REGION Network 26: *** 8 - Outputs *** Status
   #O_Status := #Status;
END_REGION

REGION Network 27: *** 8 - Outputs *** Busy
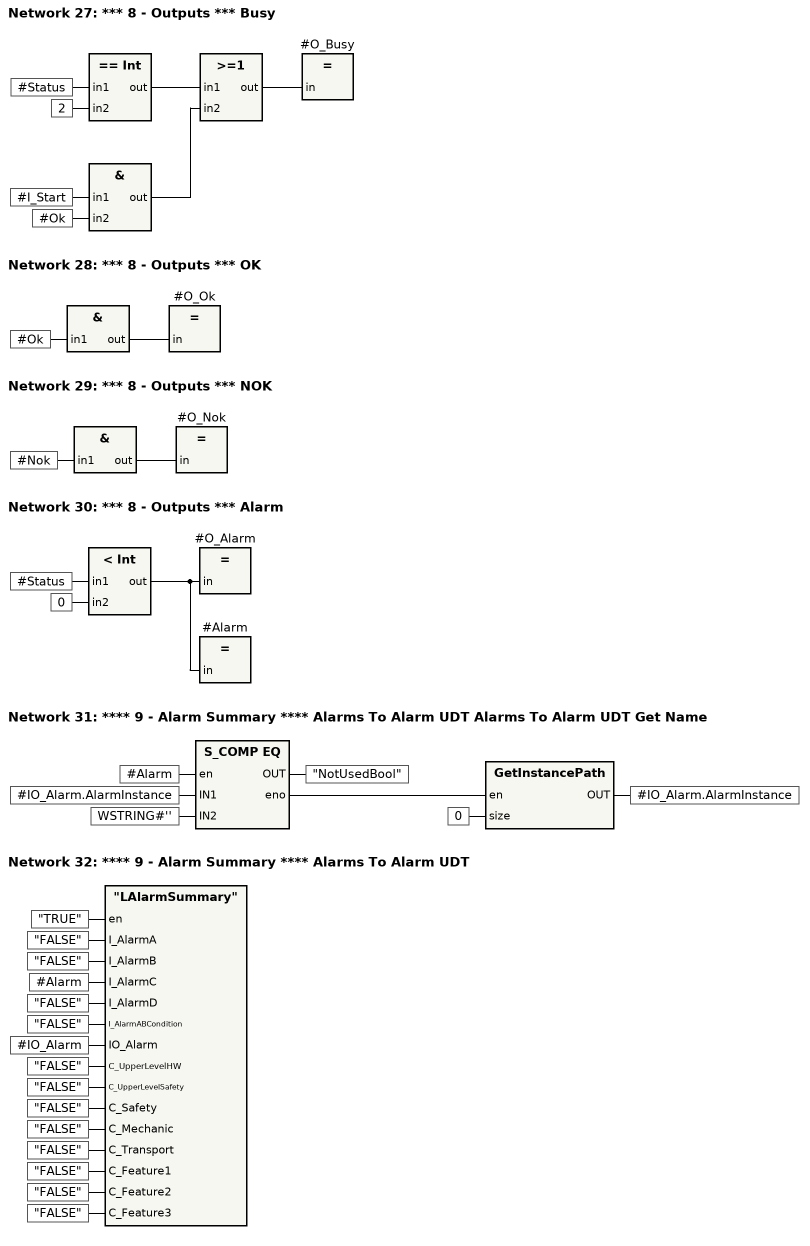
   #O_Busy := (#Status = 2) OR (#I_Start AND #Ok);
END_REGION

REGION Network 28: *** 8 - Outputs *** OK
   #O_Ok := #Ok;
END_REGION

REGION Network 29: *** 8 - Outputs *** NOK
   #O_Nok := #Nok;
END_REGION

REGION Network 30: *** 8 - Outputs *** Alarm
   #O_Alarm := #Status < 0;
   #Alarm := #O_Alarm;
END_REGION

REGION Network 31: **** 9 - Alarm Summary **** Alarms To Alarm UDT Alarms To Alarm UDT Get Name
   // Alarm / Alarm D
   S_COMP(EN := #Alarm, IN1 := #IO_Alarm.AlarmInstance, IN2 := WSTRING#'', OUT => "NotUsedBool", ENO => #_w1);
   IF #_w1 THEN GetInstancePath(size := 0, OUT => #IO_Alarm.AlarmInstance); END_IF;
END_REGION

REGION Network 32: **** 9 - Alarm Summary **** Alarms To Alarm UDT
   // Alarm / Alarm D
   IF "TRUE" THEN
       "LAlarmSummary"(I_AlarmA := "FALSE",
                       I_AlarmB := "FALSE",
                       I_AlarmC := #Alarm,
                       I_AlarmD := "FALSE",
                       I_AlarmABCondition := "FALSE",
                       IO_Alarm := #IO_Alarm,
                       C_UpperLevelHW := "FALSE",
                       C_UpperLevelSafety := "FALSE",
                       C_Safety := "FALSE",
                       C_Mechanic := "FALSE",
                       C_Transport := "FALSE",
                       C_Feature1 := "FALSE",
                       C_Feature2 := "FALSE",
                       C_Feature3 := "FALSE");
   END_IF;
END_REGION
END_FUNCTION_BLOCK

FUNCTION_BLOCK "LVIDSDeCouple"   // FB1208, SCL
{ S7_Optimized_Access := 'TRUE' }
VERSION : 0.1
// stored: AutoNumber false, IsIECCheckEnabled false, IsRetainMemResEnabled false, MemoryReserve 100, SetENOAutomatically False, UDAEnableTagReadback false
   VAR_INPUT
      C_SoftCouple { ExternalAccessible := 'False'; ExternalVisible := 'False'; ExternalWritable := 'False'} : Bool;   // If true, coupling between CarrierID and BodyID or Mixnumber, otherwise with TagID
      I_DataModeManEn { ExternalAccessible := 'False'; ExternalVisible := 'False'; ExternalWritable := 'False'} : Bool;   // Dat mode manual enabled
      I_TagID { ExternalAccessible := 'False'; ExternalVisible := 'False'; ExternalWritable := 'False'} : DWord;   // Received TagId to couple with Data / Tag ID (0 if not used)
      I_BodyID { ExternalAccessible := 'False'; ExternalVisible := 'False'; ExternalWritable := 'False'} : DWord;   // Bodynumber (0 if not used)
      I_CarrierID { ExternalAccessible := 'False'; ExternalVisible := 'False'; ExternalWritable := 'False'} : DWord;   // Carrier ID
      I_MixNbr { ExternalAccessible := 'False'; ExternalVisible := 'False'; ExternalWritable := 'False'} : DWord;   // Mixnumber (0 if not used)
      I_PopID { ExternalAccessible := 'False'; ExternalVisible := 'False'; ExternalWritable := 'False'} : UDInt;   // Spare Data / PopID (0 if not used)
      I_PopIDSuffix { ExternalAccessible := 'False'; ExternalVisible := 'False'; ExternalWritable := 'False'} : Char;   // PopID suffix (' ' if not used)
      I_PopType { ExternalAccessible := 'False'; ExternalVisible := 'False'; ExternalWritable := 'False'} : UDInt;   // Pop identifier
      I_Start { ExternalAccessible := 'False'; ExternalVisible := 'False'; ExternalWritable := 'False'} : Bool;   // Start command for coupling / Start command
   END_VAR
   VAR_OUTPUT
      O_DataModeAuto { ExternalAccessible := 'False'; ExternalVisible := 'False'; ExternalWritable := 'False'} : Bool;   // Couple or decouple in automatic mode / Data mode - Automatic
      O_DataModeMan { ExternalAccessible := 'False'; ExternalVisible := 'False'; ExternalWritable := 'False'} : Bool;   // Data mode - Manual
      O_Busy { ExternalAccessible := 'False'; ExternalVisible := 'False'; ExternalWritable := 'False'} : Bool;   // Coupling busy
      O_Status { ExternalAccessible := 'False'; ExternalVisible := 'False'; ExternalWritable := 'False'} : Int;   // Status / Status (< 0 : alarm)
      O_Alarm { ExternalAccessible := 'False'; ExternalVisible := 'False'; ExternalWritable := 'False'} : Bool;   // Alarm
      O_OK { ExternalAccessible := 'False'; ExternalVisible := 'False'; ExternalWritable := 'False'} : Bool;   // Coupling or decoupling done OK / Coupling OK
      O_NOK { ExternalAccessible := 'False'; ExternalVisible := 'False'; ExternalWritable := 'False'} : Bool;   // Coupling or decoupling done NOK / Coupling NOK
   END_VAR
   VAR_IN_OUT
      IO_VIDS : "VIDS";   // VIDS internal record
      IO_VEMData : "VEMData";   // VEM data (From master)
      IO_Alarm : "Alarm";   // Alarm
      H_DeCouple : "H_LVIDSDeCouple";
      H_HMI : "H_HMI";
   END_VAR
   VAR
      DataModeAuto { ExternalAccessible := 'False'; ExternalVisible := 'False'; ExternalWritable := 'False'} : Bool;   // Couple or decouple in automode
      DataModeAutoPls { ExternalAccessible := 'False'; ExternalVisible := 'False'; ExternalWritable := 'False'} : Bool;
      DataModeMan { ExternalAccessible := 'False'; ExternalVisible := 'False'; ExternalWritable := 'False'} : Bool;
      DataModeManPls { ExternalAccessible := 'False'; ExternalVisible := 'False'; ExternalWritable := 'False'} : Bool;
      DataModeEdit { ExternalAccessible := 'False'; ExternalVisible := 'False'; ExternalWritable := 'False'} : Bool;
      DataModeMem { ExternalAccessible := 'False'; ExternalVisible := 'False'; ExternalWritable := 'False'} : Int;
      DataModeChanged { ExternalAccessible := 'False'; ExternalVisible := 'False'; ExternalWritable := 'False'} : Bool;
      DeCoupleBeginReqPlsAuto { ExternalAccessible := 'False'; ExternalVisible := 'False'; ExternalWritable := 'False'} : Bool;
      DeCoupleBeginReqPlsMan { ExternalAccessible := 'False'; ExternalVisible := 'False'; ExternalWritable := 'False'} : Bool;
      StartPls { ExternalAccessible := 'False'; ExternalVisible := 'False'; ExternalWritable := 'False'} : Bool;
      BeginReqAuto { ExternalAccessible := 'False'; ExternalVisible := 'False'; ExternalWritable := 'False'} : Bool;
      Busy { ExternalAccessible := 'False'; ExternalVisible := 'False'; ExternalWritable := 'False'} : Bool;
      BeginReqMan { ExternalAccessible := 'False'; ExternalVisible := 'False'; ExternalWritable := 'False'} : Bool;
      CarrierID { ExternalAccessible := 'False'; ExternalVisible := 'False'; ExternalWritable := 'False'} : DWord;
      CarrierIDValid { ExternalAccessible := 'False'; ExternalVisible := 'False'; ExternalWritable := 'False'} : Bool;
   END_VAR
   VAR DB_SPECIFIC
      CarrierIDMem { ExternalAccessible := 'False'; ExternalVisible := 'False'; ExternalWritable := 'False'} : DWord;   // Memory of CarrierID at begin request
   END_VAR
   VAR
      Identification { ExternalAccessible := 'False'; ExternalVisible := 'False'; ExternalWritable := 'False'} : DWord;
      IdentificationValid { ExternalAccessible := 'False'; ExternalVisible := 'False'; ExternalWritable := 'False'} : Bool;
      IdentificationMem { ExternalAccessible := 'False'; ExternalVisible := 'False'; ExternalWritable := 'False'} : DWord;
      BodyNbr { ExternalAccessible := 'False'; ExternalVisible := 'False'; ExternalWritable := 'False'} : DWord;
      BodyNbrValid { ExternalAccessible := 'False'; ExternalVisible := 'False'; ExternalWritable := 'False'} : Bool;
      BodyIDMem { ExternalAccessible := 'False'; ExternalVisible := 'False'; ExternalWritable := 'False'} : DWord;
      MixNbr { ExternalAccessible := 'False'; ExternalVisible := 'False'; ExternalWritable := 'False'} : DWord;
      MixNbrValid { ExternalAccessible := 'False'; ExternalVisible := 'False'; ExternalWritable := 'False'} : Bool;
      MixNbrMem { ExternalAccessible := 'False'; ExternalVisible := 'False'; ExternalWritable := 'False'} : DWord;
      PopIDMem { ExternalAccessible := 'False'; ExternalVisible := 'False'; ExternalWritable := 'False'} : DWord;
      PopIDSuffixMem { ExternalAccessible := 'False'; ExternalVisible := 'False'; ExternalWritable := 'False'} : Char;
      PopTypeMem { ExternalAccessible := 'False'; ExternalVisible := 'False'; ExternalWritable := 'False'} : DWord;
      DataValid { ExternalAccessible := 'False'; ExternalVisible := 'False'; ExternalWritable := 'False'} : Bool;
      InputDataValidAuto { ExternalAccessible := 'False'; ExternalVisible := 'False'; ExternalWritable := 'False'} : Bool;
      InputDataValidMan { ExternalAccessible := 'False'; ExternalVisible := 'False'; ExternalWritable := 'False'} : Bool;
      DataNotValid { ExternalAccessible := 'False'; ExternalVisible := 'False'; ExternalWritable := 'False'} : Bool;
   END_VAR
   VAR DB_SPECIFIC
      BeginPlsModeAuto { ExternalAccessible := 'False'; ExternalVisible := 'False'; ExternalWritable := 'False'} : Bool;   // Pulse of begin in auto mode
      BeginPlsModeManTagId { ExternalAccessible := 'False'; ExternalVisible := 'False'; ExternalWritable := 'False'} : Bool;   // Pulse of begin in manual mode
      BeginReqPls { ExternalAccessible := 'False'; ExternalVisible := 'False'; ExternalWritable := 'False'} : Bool;   // Pulse of begin request
      TagIdModeManMem { ExternalAccessible := 'False'; ExternalVisible := 'False'; ExternalWritable := 'False'} : DWord;   // Memorised TagId in manual mode
      Alarm { ExternalAccessible := 'False'; ExternalVisible := 'False'; ExternalWritable := 'False'} : Bool;   // Alarm
      ChangedRcvDataAlarm { ExternalAccessible := 'False'; ExternalVisible := 'False'; ExternalWritable := 'False'} : Bool;   // Alarm received data has chnged after request
      CoupleAlarm { ExternalAccessible := 'False'; ExternalVisible := 'False'; ExternalWritable := 'False'} : Bool;   // Alarm couple or decouple NOK
      Status { ExternalAccessible := 'False'; ExternalVisible := 'False'; ExternalWritable := 'False'} : Int;   // Status
   END_VAR
   VAR
      btnDataModeAutoColour { ExternalAccessible := 'False'; ExternalVisible := 'False'; ExternalWritable := 'False'} : Word;
      btnDataModeManColour { ExternalAccessible := 'False'; ExternalVisible := 'False'; ExternalWritable := 'False'} : Word;
      btnDeCoupleVisible { ExternalAccessible := 'False'; ExternalVisible := 'False'; ExternalWritable := 'False'} : Word;
      btnDeCoupleEnable { ExternalAccessible := 'False'; ExternalVisible := 'False'; ExternalWritable := 'False'} : Word;
      btnDeCouplePls { ExternalAccessible := 'False'; ExternalVisible := 'False'; ExternalWritable := 'False'} : Bool;
      btnEditVisible { ExternalAccessible := 'False'; ExternalVisible := 'False'; ExternalWritable := 'False'} : Word;
      btnEditEnable { ExternalAccessible := 'False'; ExternalVisible := 'False'; ExternalWritable := 'False'} : Word;
      msgVEMDataBodyVisible { ExternalAccessible := 'False'; ExternalVisible := 'False'; ExternalWritable := 'False'} : Word;
      msgVEMDataCarrierVisible { ExternalAccessible := 'False'; ExternalVisible := 'False'; ExternalWritable := 'False'} : Word;
      msgDataValidVisible { ExternalAccessible := 'False'; ExternalVisible := 'False'; ExternalWritable := 'False'} : Word;   // HMI - Couple/Decouple OK
      msgDataNotValidVisible { ExternalAccessible := 'False'; ExternalVisible := 'False'; ExternalWritable := 'False'} : Word;   // HMI - Couple/Decouple OK
      msgPartPresVisible { ExternalAccessible := 'False'; ExternalVisible := 'False'; ExternalWritable := 'False'} : Word;
      txtCarrierIDDeCoupleVisible { ExternalAccessible := 'False'; ExternalVisible := 'False'; ExternalWritable := 'False'} : Word;
      txtCarrierIDDeCoupleEnable { ExternalAccessible := 'False'; ExternalVisible := 'False'; ExternalWritable := 'False'} : Word;
      txtCarrierIDDeCoupleColour { ExternalAccessible := 'False'; ExternalVisible := 'False'; ExternalWritable := 'False'} : Word;
      txtCarrierIDDeCoupleValid { ExternalAccessible := 'False'; ExternalVisible := 'False'; ExternalWritable := 'False'} : Bool;
      txtIdentificationDeCoupleVisible { ExternalAccessible := 'False'; ExternalVisible := 'False'; ExternalWritable := 'False'} : Word;
      txtIdentificationDeCoupleEnable { ExternalAccessible := 'False'; ExternalVisible := 'False'; ExternalWritable := 'False'} : Word;
      txtIdentificationDeCoupleColour { ExternalAccessible := 'False'; ExternalVisible := 'False'; ExternalWritable := 'False'} : Word;
      txtIdentificationDeCoupleValid { ExternalAccessible := 'False'; ExternalVisible := 'False'; ExternalWritable := 'False'} : Bool;
      txtMixNbrDeCoupleVisible { ExternalAccessible := 'False'; ExternalVisible := 'False'; ExternalWritable := 'False'} : Word;
      txtMixNbrDeCoupleEnable { ExternalAccessible := 'False'; ExternalVisible := 'False'; ExternalWritable := 'False'} : Word;
      txtMixNbrDeCoupleColour { ExternalAccessible := 'False'; ExternalVisible := 'False'; ExternalWritable := 'False'} : Word;
      txtMixNbrDeCoupleValid { ExternalAccessible := 'False'; ExternalVisible := 'False'; ExternalWritable := 'False'} : Bool;
      txtBodyIDDeCoupleVisible { ExternalAccessible := 'False'; ExternalVisible := 'False'; ExternalWritable := 'False'} : Word;
      txtBodyIDDeCoupleEnable { ExternalAccessible := 'False'; ExternalVisible := 'False'; ExternalWritable := 'False'} : Word;
      txtBodyIDDeCoupleColour { ExternalAccessible := 'False'; ExternalVisible := 'False'; ExternalWritable := 'False'} : Word;
      txtBodyIDDeCoupleValid { ExternalAccessible := 'False'; ExternalVisible := 'False'; ExternalWritable := 'False'} : Bool;
      txtPopIDDeCoupleVisible { ExternalAccessible := 'False'; ExternalVisible := 'False'; ExternalWritable := 'False'} : Word;
      txtPopIDDeCoupleEnable { ExternalAccessible := 'False'; ExternalVisible := 'False'; ExternalWritable := 'False'} : Word;
      txtPopIDDeCoupleColour { ExternalAccessible := 'False'; ExternalVisible := 'False'; ExternalWritable := 'False'} : Word;
      txtPopIDDeCoupleValid { ExternalAccessible := 'False'; ExternalVisible := 'False'; ExternalWritable := 'False'} : Bool;
      txtPopIDSuffixDeCoupleVisible { ExternalAccessible := 'False'; ExternalVisible := 'False'; ExternalWritable := 'False'} : Word;
      txtPopIDSuffixDeCoupleEnable { ExternalAccessible := 'False'; ExternalVisible := 'False'; ExternalWritable := 'False'} : Word;
      txtPopIDSuffixDeCoupleColour { ExternalAccessible := 'False'; ExternalVisible := 'False'; ExternalWritable := 'False'} : Word;
      txtPopTypeDeCoupleVisible { ExternalAccessible := 'False'; ExternalVisible := 'False'; ExternalWritable := 'False'} : Word;
      txtPopTypeDeCoupleEnable { ExternalAccessible := 'False'; ExternalVisible := 'False'; ExternalWritable := 'False'} : Word;
      txtPopTypeDeCoupleColour { ExternalAccessible := 'False'; ExternalVisible := 'False'; ExternalWritable := 'False'} : Word;
      IconColour { ExternalAccessible := 'False'; ExternalVisible := 'False'; ExternalWritable := 'False'} : Word;
      DeCoupleOK { ExternalAccessible := 'False'; ExternalVisible := 'False'; ExternalWritable := 'False'} : Bool;
      DeCoupleNOK { ExternalAccessible := 'False'; ExternalVisible := 'False'; ExternalWritable := 'False'} : Bool;
      _DataModeManForcedPls { ExternalAccessible := 'False'; ExternalVisible := 'False'; ExternalWritable := 'False'; S7_SetPoint := 'True'} : R_TRIG;
      _DataModeAutoPls { ExternalAccessible := 'False'; ExternalVisible := 'False'; ExternalWritable := 'False'; S7_SetPoint := 'True'} : R_TRIG;
      _DeCoupleStartPls { ExternalAccessible := 'False'; ExternalVisible := 'False'; ExternalWritable := 'False'; S7_SetPoint := 'True'} : R_TRIG;
      _DataModeChangedPls { ExternalAccessible := 'False'; ExternalVisible := 'False'; ExternalWritable := 'False'; S7_SetPoint := 'True'} : R_TRIG;
      _btnDeCouplePls { ExternalAccessible := 'False'; ExternalVisible := 'False'; ExternalWritable := 'False'; S7_SetPoint := 'True'} : R_TRIG;
   END_VAR
   VAR CONSTANT
      STATUS_OK : Int := 1;
      STATUS_COUPLE_REQ : Int := 107;
      STATUS_COUPLE_RUNNING : Int := 207;
      STATUS_DECOUPLE_REQ : Int := 108;
      STATUS_DECOUPLE_RUNNING : Int := 208;
      OFF : Word := 2#0000000000000000;
      ON : Word := 2#0000000000000001;
      VISIBLE : Word := 2#0000000000000001;
      ENABLE : Word := 2#0000000000000010;
      BG_COLOUR_GREY : Word := 2#0000000000000100;
      COLOUR_DEFAULT : Word := 2#0000000000000000;
      COLOUR_RED : Word := 2#0000000000010000;
      COLOUR_GREEN : Word := 2#0000000000100000;
      COLOUR_BLUE : Word := 2#0000000001000000;
      COLOUR_WHITE : Word := 2#0000000010000000;
      BG_COLOUR_BLUE_FLASH : Word := 2#0000000010000000;
      BG_COLOUR_LIGHTRED : Word := 2#0100000000000000;
      BG_COLOUR_YELLOW : Word := 2#1000000000000000;
      OK_BEGIN_DELAY_MAX : Time := T#10s;
      CMD_DECOUPLE : DWord := 2006;
   END_VAR
BEGIN
   (******************************************************************************)
   (* Data mode - Activation                                                     *)
   (******************************************************************************)

   //Automatic
   //Data mode selected  - No mode, select auto
   IF (#H_DeCouple.H_selDataMode < 1) OR (#H_DeCouple.H_selDataMode > 3) OR NOT #IO_VIDS.PartPres OR NOT #I_DataModeManEn THEN
       #H_DeCouple.H_selDataMode := 1;
   END_IF;

   //Data mode automatic - Activation
   #DataModeAuto := (#H_DeCouple.H_selDataMode = 1);

   //Data mode automatic - Create pulse upon selection 
   #_DataModeAutoPls(CLK:=#DataModeAuto,Q=>#DataModeAutoPls);

   //Data mode manual - Activation
   #DataModeMan := (#H_DeCouple.H_selDataMode = 2);

   //Data mode manual - Create pulse upon selection
   #_DataModeManForcedPls(CLK := #DataModeMan,Q => #DataModeManPls);

   //Data mode changed
   #_DataModeAutoPls(CLK := #H_DeCouple.H_selDataMode <> #DataModeMem,Q => #DataModeAutoPls);
   #DataModeMem:=#H_DeCouple.H_selDataMode;

   //Data mode edit - Activation
   IF #DataModeMan AND (#H_DeCouple.H_btnEdit = #ON) THEN
       #DataModeEdit := TRUE;
       //Copy VEM data to HMI
       #H_DeCouple.H_txtIdentification := #IO_VEMData.Identification;

   ELSIF #DataModeAuto THEN
       #DataModeEdit := FALSE;
   END_IF;


   IF #DataModeEdit THEN

       //Check valid
       #txtCarrierIDDeCoupleValid := #H_DeCouple.H_txtCarrierIDDeCouple > 0;
       #txtIdentificationDeCoupleValid := #H_DeCouple.H_txtIdentificationDeCouple > 0;
       #txtBodyIDDeCoupleValid :=#H_DeCouple.H_txtBodyIDDeCouple > 0;
       #txtMixNbrDeCoupleValid := #H_DeCouple.H_txtMixNbrDeCouple > 0;
       #txtPopIDDeCoupleValid := #H_DeCouple.H_txtPopIdDeCouple > 0;

       //Entry fields valid
       #InputDataValidMan := #txtCarrierIDDeCoupleValid AND (#txtIdentificationDeCoupleValid OR #txtBodyIDDeCoupleValid OR #txtMixNbrDeCoupleValid OR #txtPopIDDeCoupleValid);

   ELSE

       //Reset
       #InputDataValidMan := FALSE;

   END_IF;

   (******************************************************************************)
   (* Data mode automatic - Begin request                                        *)
   (******************************************************************************)

   //Start - Create pulse
   #_DeCoupleStartPls(CLK := #I_Start,
                    Q => #StartPls);

   #BeginReqAuto:=False;
   IF #DataModeAuto AND #StartPls AND #IO_VIDS.PartPres AND #I_CarrierID > 0  THEN

       //Memorize parameters
       #IdentificationMem := #I_TagID;
       #BodyIDMem := #I_BodyID;
       #CarrierIDMem := #I_CarrierID;
       #MixNbrMem := #I_MixNbr;
       #PopIDMem := #I_PopID;
       #PopIDSuffixMem := #I_PopIDSuffix;
       #PopTypeMem := #I_PopType;

       //Data mode automatic - Begin request
       #BeginReqAuto := True;

   END_IF;

   (******************************************************************************)
   (* Data mode manual - Begin request                                           *)
   (******************************************************************************)

   //Couple button - Create pulse 
   #_btnDeCouplePls(CLK:=#H_DeCouple.H_btnDecouple=#ON,
                  Q=>#btnDeCouplePls);

   #BeginReqMan := False;
   IF #DataModeEdit AND #btnDeCouplePls AND #IO_VIDS.PartPres THEN

       //Edit mode off
       #DataModeEdit := FALSE;

       //Memorize data
       #CarrierIDMem := #H_DeCouple.H_txtCarrierIDDeCouple;

       //Start with a clean sheet
       #IdentificationMem := 0;
       #BodyIDMem := 0;
       #MixNbrMem := 0;
       #PopIDMem := 0;
       #PopIDSuffixMem := ' ';
       #PopTypeMem := 0;

       //Memorize parameters
       IF #H_DeCouple.H_txtIdentificationDeCouple > 0 THEN
           #IdentificationMem := #H_DeCouple.H_txtIdentificationDeCouple;
       ELSIF #H_DeCouple.H_txtBodyIDDeCouple > 0 THEN
           #BodyIDMem := #H_DeCouple.H_txtBodyIDDeCouple;
       ELSIF #H_DeCouple.H_txtMixNbrDeCouple > 0 THEN
           #MixNbrMem := #H_DeCouple.H_txtMixNbrDeCouple;
       ELSIF #H_DeCouple.H_txtPopIdDeCouple > 0 OR #H_DeCouple.H_txtPopIdSuffixDeCouple <> ' ' OR #H_DeCouple.H_txtPopTypeDeCouple <> 0  THEN
           #PopIDMem := #H_DeCouple.H_txtPopIdDeCouple;
           #PopIDSuffixMem := #H_DeCouple.H_txtPopIdSuffixDeCouple;
           #PopTypeMem := #H_DeCouple.H_txtPopTypeDeCouple;
       END_IF;

       //Data mode manual - begin request
       #BeginReqMan := True;

   END_IF;

   (******************************************************************************)
   (* Begin request - Summary                                                    *)
   (******************************************************************************)

   #IO_VIDS.DeCouple.BeginReq := #BeginReqAuto OR #BeginReqMan;

   IF #IO_VIDS.DeCouple.BeginReq THEN
       #DeCoupleOK := False;
       #DeCoupleNOK := False;
   END_IF;

   (*******************************************************)
   (* Begin                                               *)
   (*******************************************************)

   IF #IO_VIDS.DeCouple.OkBegin THEN
       //Initialize parameters
       #IO_VIDS.VEMData.IdType := #IO_VIDS.IDType;
       #IO_VIDS.VEMData.FunctionCode := 255;
       #IO_VIDS.VEMData.Identification := #IdentificationMem;
       #IO_VIDS.VEMData.BodyID := #BodyIDMem;
       #IO_VIDS.VEMData.CarrierID := #CarrierIDMem;
       #IO_VIDS.VEMData.MixNumber := #MixNbrMem;
       #IO_VIDS.VEMData.PopID := #PopIDMem;
       #IO_VIDS.VEMData.PopIDSuffix := #PopIDSuffixMem;
       #IO_VIDS.VEMData.PopType := #PopTypeMem;
       #IO_VIDS.VEMData.CommandCode := #CMD_DECOUPLE;
       #Status := #IO_VIDS.DeCouple.Status;
   END_IF;

   #IO_VIDS.DeCouple.Begin := #IO_VIDS.DeCouple.OkBegin;

   (*******************************************************)
   (* Running                                             *)
   (*******************************************************)
   IF #IO_VIDS.DeCouple.Running THEN
       #Status := #IO_VIDS.DeCouple.Status;
   END_IF;

   #Busy := #IO_VIDS.DeCouple.Running;

   (*******************************************************)
   (* Finish                                              *)
   (*******************************************************)

   IF #IO_VIDS.DeCouple.Finished THEN

       //Update status
       #Status := #IO_VIDS.DeCouple.Status;

       //Status OK/NOK
       IF #Status = #STATUS_OK THEN
           #DeCoupleOK := True;
       ELSE
           #DeCoupleNOK := True;
           IF #DataModeMan THEN
               #DataModeEdit := TRUE;
           END_IF;
       END_IF;

   END_IF;

   (******************************************************************************)
   (* Alarm                                                                      *)
   (******************************************************************************)

   #Alarm := (#Status < 0);

   "LAlarmSummary"(I_AlarmA := "FALSE",
                   I_AlarmB := "FALSE",
                   I_AlarmC := #Alarm,
                   I_AlarmD := "FALSE",
                   I_AlarmABCondition := "FALSE",
                   IO_Alarm := #IO_Alarm,
                   C_UpperLevelHW := "FALSE",
                   C_UpperLevelSafety := "FALSE",
                   C_Safety := "FALSE",
                   C_Mechanic := "FALSE",
                   C_Transport := "FALSE",
                   C_Feature1 := "FALSE",
                   C_Feature2 := "FALSE",
                   C_Feature3 := "FALSE");


   (*******************************************************)
   (* Reset                                               *)
   (*******************************************************)

   IF NOT #IO_VIDS.PartPres THEN
       #DeCoupleOK := False;
       #DeCoupleNOK := False;
       #H_DeCouple.H_txtIdentification := 0;
       #H_DeCouple.H_txtBodyID := 0;
       #H_DeCouple.H_txtCarrierID := 0;
       #H_DeCouple.H_txtMixNbr := 0;
       #H_DeCouple.H_txtPopId := 0;
       #H_DeCouple.H_txtPopIdSuffix := ' ';
       #H_DeCouple.H_txtPopType := 0;
       #Status := 0;
   END_IF;

   (*******************************************************)
   (* Outputs                                             *)
   (*******************************************************)

   #O_DataModeAuto := #DataModeAuto;
   #O_DataModeMan := #DataModeMan;
   #O_OK := #DeCoupleOK;
   #O_NOK := #DeCoupleNOK;

   #O_Busy := #Busy;
   #O_Status := #Status;
   #O_Alarm := #Status < 0;

   (*******************************************************)
   (* HMI - Reset buttons                                 *)
   (*******************************************************)

   #H_DeCouple.H_btnEdit := #OFF;
   #H_DeCouple.H_btnDecouple := #OFF;
   #H_DeCouple.H_btnDecouple := #OFF;

   (*******************************************************)
   (* HMI - Update text fields                            *)
   (*******************************************************)

   IF #IO_VIDS.VEMDataValid THEN
       #H_DeCouple.H_txtCarrierIDDeCouple := #IO_VEMData.CarrierID;
       #H_DeCouple.H_txtIdentificationDeCouple := #IO_VEMData.Identification;
       #H_DeCouple.H_txtBodyIDDeCouple := #IO_VEMData.BodyID;
       #H_DeCouple.H_txtMixNbrDeCouple := #IO_VEMData.MixNumber;
       #H_DeCouple.H_txtPopId := #IO_VEMData.PopID;
       #H_DeCouple.H_txtPopIdSuffix := #IO_VEMData.PopIDSuffix;
       #H_DeCouple.H_txtPopType := #IO_VEMData.PopType;
   ELSE
       #H_DeCouple.H_txtCarrierID := 0;
       #H_DeCouple.H_txtIdentification := 0;
       #H_DeCouple.H_txtBodyID := 0;
       #H_DeCouple.H_txtMixNbr := 0;
       #H_DeCouple.H_txtPopId := 0;
       #H_DeCouple.H_txtPopIdSuffix := ' ';
       #H_DeCouple.H_txtPopType := 0;
   END_IF;

   (*******************************************************)
   (* HMI - Input fields                                  *)
   (*******************************************************)

   //Visible
   #txtIdentificationDeCoupleVisible := #OFF;
   #txtBodyIDDeCoupleVisible := #OFF;
   #txtCarrierIDDeCoupleVisible := #OFF;
   #txtMixNbrDeCoupleVisible := #OFF;
   #txtPopIDDeCoupleVisible := #OFF;
   #txtPopIDSuffixDeCoupleVisible := #OFF;
   #txtPopTypeDeCoupleVisible := #OFF;

   IF #DataModeMan THEN
       #txtCarrierIDDeCoupleVisible := #VISIBLE;
       IF #C_SoftCouple THEN
           #txtBodyIDDeCoupleVisible := #VISIBLE;
           #txtMixNbrDeCoupleVisible := #VISIBLE;
           #txtPopIDDeCoupleVisible := #VISIBLE;
           #txtPopIDSuffixDeCoupleVisible := #VISIBLE;
           #txtPopTypeDeCoupleVisible := #VISIBLE;
       ELSE
           #txtIdentificationDeCoupleVisible := #VISIBLE;
       END_IF;
   END_IF;

   //Enable
   #txtIdentificationDeCoupleEnable := #OFF;
   #txtCarrierIDDeCoupleEnable := #OFF;
   #txtBodyIDDeCoupleEnable := #OFF;
   #txtMixNbrDeCoupleEnable := #OFF;
   #txtPopIDDeCoupleEnable := #OFF;
   #txtPopIDSuffixDeCoupleEnable := #OFF;
   #txtPopTypeDeCoupleEnable := #OFF;

   IF #DataModeEdit THEN
       #txtCarrierIDDeCoupleEnable := #ENABLE;
       IF #C_SoftCouple THEN
           #txtBodyIDDeCoupleEnable := #ENABLE;
           #txtMixNbrDeCoupleEnable := #ENABLE;
           #txtPopIDDeCoupleEnable := #ENABLE;
           #txtPopIDSuffixDeCoupleEnable := #ENABLE;
           #txtPopTypeDeCoupleEnable := #ENABLE;
       ELSE
           #txtIdentificationDeCoupleEnable := #ENABLE;
       END_IF;
   END_IF;

   (*******************************************************)
   (* HMI - Buttons                                       *)
   (*******************************************************)

   //HMI - Button Data mode automatic
   IF #DataModeAuto THEN
       #btnDataModeAutoColour := #COLOUR_GREEN;
   ELSE
       #btnDataModeAutoColour := #COLOUR_DEFAULT;
   END_IF;

   //HMI - Button Data mode manual
   IF #DataModeMan THEN
       #btnDataModeManColour := #COLOUR_BLUE;
   ELSE
       #btnDataModeManColour := #COLOUR_DEFAULT;
   END_IF;

   //HMI - Button Edit
   IF #DataModeMan AND NOT #DataModeEdit AND NOT #IO_VIDS.Couple.Running THEN
       #btnEditVisible := #VISIBLE;
       #btnEditEnable := #ENABLE;
   ELSE
       #btnEditVisible := #OFF;
       #btnEditEnable := #OFF;
   END_IF;

   //HMI - Button Couple
   IF #DataModeEdit AND #InputDataValidMan THEN
       #btnDeCoupleVisible := #VISIBLE;
       #btnDeCoupleEnable := #ENABLE;
   ELSE
       #btnDeCoupleVisible := #OFF;
       #btnDeCoupleEnable := #OFF;
   END_IF;

   (*******************************************************)
   (* HMI - Messages                                      *)
   (*******************************************************)

   //HMI - Message part present
   IF #IO_VIDS.PartPres THEN
       #msgPartPresVisible := #VISIBLE;
   ELSE
       #msgPartPresVisible := #OFF;
   END_IF;

   //HMI - Message data valid, not valid
   IF #IO_VIDS.VEMDataValid THEN
       #msgDataValidVisible := #VISIBLE;
   ELSIF #IO_VIDS.VEMDataNotValid THEN
       #msgDataNotValidVisible := #VISIBLE;
   ELSE
       #msgDataValidVisible := #OFF;
       #msgDataNotValidVisible := #OFF;
   END_IF;

   //Body or carrier data
   IF #IO_VIDS.IDType = 0 THEN
       #msgVEMDataBodyVisible := #VISIBLE;
       #msgVEMDataCarrierVisible := #OFF;
   ELSE
       #msgVEMDataBodyVisible := #OFF;
       #msgVEMDataCarrierVisible := #VISIBLE;
   END_IF;

   (*******************************************************)
   (* Icon - animation                                    *)
   (*******************************************************)

   "LIAnimDWord"(I_SetPos:=FALSE,
                   I_ResetPos:=FALSE,
                   I_Active:=#Status>1,
                   I_Visible:=FALSE,
                   I_OutOfUse:=FALSE,
                   I_IntlkSet:=FALSE,
                   I_IntlkReset:=FALSE,
                   I_IntlkSetAlm:=FALSE,
                   I_IntlkResetAlm:=FALSE,
                   I_ManualMode:=#DataModeMan,
                   I_FncSelInHMI:=FALSE,
                   I_AnySelected:=FALSE,
                   I_AlarmA:=FALSE,
                   I_AlarmB:=FALSE,
                   I_AlarmC:=#Status<0,
                   I_AlarmD:=FALSE,
                   I_SafetyOk:=FALSE,
                   I_Service:="TRUE",
                 I_Spare1:="FALSE",
                 I_Spare2:="FALSE",
                 I_Spare3:="FALSE",
                 I_Spare4:="FALSE",
                 I_Spare5:="FALSE",
                 I_Spare6:="FALSE",
                 I_Spare7:="FALSE",
                 I_Spare8:="FALSE",
                 I_Spare9:="FALSE",
                 I_Spare10:="FALSE",
                 I_Spare11:="FALSE",
                 I_Spare12:="FALSE",
                 I_Spare13:="FALSE",
                 I_Spare14:="FALSE",
                 H_IAnim=>#H_HMI.H_IAnim);

   (*******************************************************)
   (* HMI - Animations summary                            *)
   (*******************************************************)

   #H_DeCouple.H_txtCommandCodeSent := #IO_VIDS.CmdCodeSent;
   #H_DeCouple.H_txtCommandCodeRcvd := #IO_VIDS.CmdCodeRcvd;
   #H_DeCouple.H_msgVEMDataBodyAnim := #msgVEMDataBodyVisible;
   #H_DeCouple.H_msgVEMDataCarrierAnim := #msgVEMDataCarrierVisible;
   #H_DeCouple.H_btnDataModeAutoAnim := #btnDataModeAutoColour;
   #H_DeCouple.H_btnDataModeManAnim := #btnDataModeManColour;
   #H_DeCouple.H_txtCarrierIDDeCoupleAnim := #txtCarrierIDDeCoupleVisible OR #txtCarrierIDDeCoupleEnable OR #txtCarrierIDDeCoupleColour;
   #H_DeCouple.H_txtIdentificationDeCoupleAnim := #txtIdentificationDeCoupleVisible OR #txtIdentificationDeCoupleEnable OR #txtIdentificationDeCoupleColour;
   #H_DeCouple.H_txtBodyIDDeCoupleAnim := #txtBodyIDDeCoupleVisible OR #txtBodyIDDeCoupleEnable OR #txtBodyIDDeCoupleColour;
   #H_DeCouple.H_txtMixNbrDeCoupleAnim := #txtMixNbrDeCoupleVisible OR #txtMixNbrDeCoupleEnable OR #txtMixNbrDeCoupleColour;
   #H_DeCouple.H_txtPopIdDeCoupleAnim := #txtPopIDDeCoupleVisible OR #txtPopIDDeCoupleEnable OR #txtPopIDDeCoupleColour;
   #H_DeCouple.H_txtPopIdSuffixDeCoupleAnim := #txtPopIDSuffixDeCoupleVisible OR #txtPopIDSuffixDeCoupleEnable OR #txtPopIDSuffixDeCoupleColour;
   #H_DeCouple.H_txtPopTypeDeCoupleAnim := #txtPopTypeDeCoupleVisible OR #txtPopTypeDeCoupleEnable OR #txtPopTypeDeCoupleColour;
   #H_DeCouple.H_btnEditAnim := #btnEditVisible OR #btnEditEnable;
   #H_DeCouple.H_btnDecoupleAnim := #btnDeCoupleVisible OR #btnDeCoupleEnable;
   #H_DeCouple.H_msgPartPresAnim := #msgPartPresVisible;
   #H_DeCouple.H_msgVEMDataValidAnim := #msgDataValidVisible;
   #H_DeCouple.H_msgVEMDataNotValidAnim := #msgDataNotValidVisible;
   #H_DeCouple.H_msgStatus := #Status;
END_FUNCTION_BLOCK

FUNCTION_BLOCK "LVIDSQualityRequest"   // FB1220, SCL
{ S7_Optimized_Access := 'TRUE' }
VERSION : 0.1
// stored: AutoNumber false, IsIECCheckEnabled false, IsRetainMemResEnabled false, MemoryReserve 100, SetENOAutomatically False, UDAEnableTagReadback false
   VAR_INPUT
      I_TagID { ExternalAccessible := 'False'; ExternalVisible := 'False'; ExternalWritable := 'False'} : DWord;   // Tag ID
      I_BodyID { ExternalAccessible := 'False'; ExternalVisible := 'False'; ExternalWritable := 'False'} : DWord;   // Body ID
      I_CarrierID { ExternalAccessible := 'False'; ExternalVisible := 'False'; ExternalWritable := 'False'} : DWord;   // Carrier ID
      I_MixNr { ExternalAccessible := 'False'; ExternalVisible := 'False'; ExternalWritable := 'False'} : DWord;   // Mix Nr
      I_PopID { ExternalAccessible := 'False'; ExternalVisible := 'False'; ExternalWritable := 'False'} : UDInt;   // Spare Data / PopID
      I_PopIDSuffix { ExternalAccessible := 'False'; ExternalVisible := 'False'; ExternalWritable := 'False'} : Char;   // PopID suffix
      I_PopType { ExternalAccessible := 'False'; ExternalVisible := 'False'; ExternalWritable := 'False'} : UDInt;   // Pop identifier
      I_ManualModeVisible { ExternalAccessible := 'False'; ExternalVisible := 'False'; ExternalWritable := 'False'} : Bool := 0;   // 0= Hidden 1= Visible
      I_Start { ExternalAccessible := 'False'; ExternalVisible := 'False'; ExternalWritable := 'False'} : Bool;   // Start command
   END_VAR
   VAR_OUTPUT
      O_DataModeAuto { ExternalAccessible := 'False'; ExternalVisible := 'False'; ExternalWritable := 'False'} : Bool;   // Data mode - Automatic
      O_DataModeMan { ExternalAccessible := 'False'; ExternalVisible := 'False'; ExternalWritable := 'False'} : Bool;   // Data mode - Manual
      O_DataValid { ExternalAccessible := 'False'; ExternalVisible := 'False'; ExternalWritable := 'False'} : Bool;   // Data valid
      O_DataNotValid { ExternalAccessible := 'False'; ExternalVisible := 'False'; ExternalWritable := 'False'} : Bool;   // Data not valid
      O_BodyCargoStatusOk { ExternalAccessible := 'False'; ExternalVisible := 'False'; ExternalWritable := 'False'} : Bool;
      O_BodyCargoStatusNok { ExternalAccessible := 'False'; ExternalVisible := 'False'; ExternalWritable := 'False'} : Bool;
      O_Busy { ExternalAccessible := 'False'; ExternalVisible := 'False'; ExternalWritable := 'False'} : Bool;   // Busy
      O_Status { ExternalAccessible := 'False'; ExternalVisible := 'False'; ExternalWritable := 'False'} : Int;   // Status code
      O_Alarm { ExternalAccessible := 'False'; ExternalVisible := 'False'; ExternalWritable := 'False'} : Bool;   // Alarm
      O_VemData { ExternalAccessible := 'False'; ExternalVisible := 'False'; ExternalWritable := 'False'} : "VEMData";
   END_VAR
   VAR_IN_OUT
      IO_VIDS : "VIDS";   // PCS data record
      IO_Alarm : "Alarm";   // Alarm
      H_HMI : "H_HMI";
      H_LVIDSQualityRequest : "H_LVIDSQualityRequest";   // HMI - specific interface
   END_VAR
   VAR
      DataModeAuto { ExternalAccessible := 'False'; ExternalVisible := 'False'; ExternalWritable := 'False'} : Bool;
      DataModeAutoEdge { ExternalAccessible := 'False'; ExternalVisible := 'False'; ExternalWritable := 'False'} : Bool;
      DataModeAutoPls { ExternalAccessible := 'False'; ExternalVisible := 'False'; ExternalWritable := 'False'} : Bool;
      DataModeMan { ExternalAccessible := 'False'; ExternalVisible := 'False'; ExternalWritable := 'False'} : Bool;
      DataModeManEdge { ExternalAccessible := 'False'; ExternalVisible := 'False'; ExternalWritable := 'False'} : Bool;
      DataModeManPls { ExternalAccessible := 'False'; ExternalVisible := 'False'; ExternalWritable := 'False'} : Bool;
      DataModeChanged { ExternalAccessible := 'False'; ExternalVisible := 'False'; ExternalWritable := 'False'} : Bool;
      StartCmdEdgAuto { ExternalAccessible := 'False'; ExternalVisible := 'False'; ExternalWritable := 'False'} : Bool;
      StartCmdPlsAuto { ExternalAccessible := 'False'; ExternalVisible := 'False'; ExternalWritable := 'False'} : Bool;
      StartCmdPlsMan { ExternalAccessible := 'False'; ExternalVisible := 'False'; ExternalWritable := 'False'} : Bool;
      StartCmdEdgMan { ExternalAccessible := 'False'; ExternalVisible := 'False'; ExternalWritable := 'False'} : Bool;
      BeginReqPlsDataModeAuto { ExternalAccessible := 'False'; ExternalVisible := 'False'; ExternalWritable := 'False'} : Bool;
      BeginReqPlsDataModeMan { ExternalAccessible := 'False'; ExternalVisible := 'False'; ExternalWritable := 'False'} : Bool;
      Status { ExternalAccessible := 'False'; ExternalVisible := 'False'; ExternalWritable := 'False'} : Int;
      BtnModeManConfirm { ExternalAccessible := 'False'; ExternalVisible := 'False'; ExternalWritable := 'False'} : Bool;
      Alarm { ExternalAccessible := 'False'; ExternalVisible := 'False'; ExternalWritable := 'False'} : Bool;
      DataValid { ExternalAccessible := 'False'; ExternalVisible := 'False'; ExternalWritable := 'False'} : Bool;
      DataNotValid { ExternalAccessible := 'False'; ExternalVisible := 'False'; ExternalWritable := 'False'} : Bool;
      TagIDMem { ExternalAccessible := 'False'; ExternalVisible := 'False'; ExternalWritable := 'False'} : DWord;
      BodyIDMem { ExternalAccessible := 'False'; ExternalVisible := 'False'; ExternalWritable := 'False'} : DWord;
      CarrierIDMem { ExternalAccessible := 'False'; ExternalVisible := 'False'; ExternalWritable := 'False'} : DWord;
      MixNrMem { ExternalAccessible := 'False'; ExternalVisible := 'False'; ExternalWritable := 'False'} : DWord;
      PopIDMem { ExternalAccessible := 'False'; ExternalVisible := 'False'; ExternalWritable := 'False'} : UDInt;
      PopIDSuffixMem { ExternalAccessible := 'False'; ExternalVisible := 'False'; ExternalWritable := 'False'} : Char;
      PopTypeMem { ExternalAccessible := 'False'; ExternalVisible := 'False'; ExternalWritable := 'False'} : UDInt;
      BodyCargoStatusOk { ExternalAccessible := 'False'; ExternalVisible := 'False'; ExternalWritable := 'False'} : Bool;
      BodyCargoStatusNok { ExternalAccessible := 'False'; ExternalVisible := 'False'; ExternalWritable := 'False'} : Bool;
      BodyType1 { ExternalAccessible := 'False'; ExternalVisible := 'False'; ExternalWritable := 'False'} : DWord;
      VemData { ExternalAccessible := 'False'; ExternalVisible := 'False'; ExternalWritable := 'False'; S7_SetPoint := 'True'} : "VEMData";
      VemDataEmty { ExternalAccessible := 'False'; ExternalVisible := 'False'; ExternalWritable := 'False'; S7_SetPoint := 'True'} : "VEMData";
      H_btnConfirmDataModeManEnable : Word;
      H_btnConfirmDataModeManVisible : Word;
      H_txtSequenceNrEnable : Word;
      H_txtSequenceNrVisible : Word;
      H_txtSequenceNrColour : Word;
      H_txtFieldBodyType1Color : Word;
      H_txtFieldBodyType1Visible : Word;
      H_txtFieldBodyType1Enable : Word;
   END_VAR
   VAR_TEMP
      Temp_NotUsedBool : Bool;
   END_VAR
   VAR CONSTANT
      C_Command : DWord := 3041;   // Command for specific data
      OFF : Word := 2#0000000000000000;
      ENABLE : Word := 2#0000000000000001;
      VISIBLE : Word := 2#0000000000000010;
      COLOUR_GREY : Word := 2#0000000000010000;
      COLOUR_WHITE : Word := 2#0000000000100000;
      COLOUR_GREEN : Word := 2#0000000001000000;
      COLOUR_RED : Word := 2#0000000010000000;
      COLOUR_BLUE_FLASH : Word := 2#0000000100000000;
   END_VAR
BEGIN
   (******************************************************************************************  
    Changelog

       2017/06/21 AndriesHeynssens
       - Module 5005 based on the module GetSpecData build by PMo

    Description

       This module gets specific cardata from production server
       Adapt the following sections to your needs :

           IT Code 3041 Atacq

    List of authors

       Company : Volvo Cars Gent
       Name    : Patrick Moreau (PMo)
       E-mail  : patrick.moreau@volvocars.com
       Tel.    : +32 9 2503165

    ******************************************************************************************)


   (******************************************************************************)
   (* Input from HMI - Buttons                                                   *)
   (******************************************************************************)
   // FC1014
   "LDWordToBit"(I_DWord:=#H_HMI.H_CommandDW1,
                 O_0=>#BtnModeManConfirm,
                 O_1=>#Temp_NotUsedBool,
                 O_2=>#Temp_NotUsedBool,
                 O_3=>#Temp_NotUsedBool,
                 O_4=>#Temp_NotUsedBool,
                 O_5=>#Temp_NotUsedBool,
                 O_6=>#Temp_NotUsedBool,
                 O_7=>#Temp_NotUsedBool,
                 O_8=>#Temp_NotUsedBool,
                 O_9=>#Temp_NotUsedBool,
                 O_10=>#Temp_NotUsedBool,
                 O_11=>#Temp_NotUsedBool,
                 O_12=>#Temp_NotUsedBool,
                 O_13=>#Temp_NotUsedBool,
                 O_14=>#Temp_NotUsedBool,
                 O_15=>#Temp_NotUsedBool,
                 O_16=>#Temp_NotUsedBool,
                 O_17=>#Temp_NotUsedBool,
                 O_18=>#Temp_NotUsedBool,
                 O_19=>#Temp_NotUsedBool,
                 O_20=>#Temp_NotUsedBool,
                 O_21=>#Temp_NotUsedBool,
                 O_22=>#Temp_NotUsedBool,
                 O_23=>#Temp_NotUsedBool,
                 O_24=>#Temp_NotUsedBool,
                 O_25=>#Temp_NotUsedBool,
                 O_26=>#Temp_NotUsedBool,
                 O_27=>#Temp_NotUsedBool,
                 O_28=>#Temp_NotUsedBool,
                 O_29=>#Temp_NotUsedBool,
                 O_30=>#Temp_NotUsedBool,
                 O_31=>#Temp_NotUsedBool);
   #H_HMI.H_CommandDW1 := 0;

   (******************************************************************************)
   (* Data mode - Automatic                                                      *)
   (******************************************************************************)  
   //Data mode selected  - No mode, select auto
   IF (#H_LVIDSQualityRequest.H_selDataMode < 1) OR (#H_LVIDSQualityRequest.H_selDataMode > 2) OR NOT #IO_VIDS.PartPres  THEN
       #H_LVIDSQualityRequest.H_selDataMode := 1;
   END_IF;

   #DataModeAuto:=(#H_LVIDSQualityRequest.H_selDataMode=1);
   #DataModeAutoPls := #DataModeAuto AND NOT #DataModeAutoEdge;
   #DataModeAutoEdge := #DataModeAuto;

   (******************************************************************************)
   (* Data mode - Manual                                                         *)
   (******************************************************************************)
   #DataModeMan := (#H_LVIDSQualityRequest.H_selDataMode = 2);
   #DataModeManPls := #DataModeMan AND NOT #DataModeManEdge;
   #DataModeManEdge := #DataModeMan;

   (******************************************************************************)
   (* Data mode - SIMULATE                                                       *)
   (******************************************************************************)

   //Data mode changed
   #DataModeChanged := #DataModeAutoPls OR #DataModeManPls;

   (******************************************************************************************************************************)
   (* COMMUNICATION WITH IT                                                                                                      *)
   (******************************************************************************************************************************)

   (******************************************************************************)
   (* Start Pulses                                                               *)
   (******************************************************************************)
   //Start command pulse - Data mode automatic
   #StartCmdPlsAuto := #I_Start AND NOT #StartCmdEdgAuto;
   #StartCmdEdgAuto := #I_Start;

   //Start command pulse - Data mode manual
   #StartCmdPlsMan := #BtnModeManConfirm AND NOT #StartCmdEdgMan;    
   #StartCmdEdgMan := #BtnModeManConfirm;

   (******************************************************************************)
   (* Begin request                                                              *)
   (******************************************************************************)

   //Begin request
   #BeginReqPlsDataModeAuto := (#StartCmdPlsAuto AND #DataModeAuto);
   #BeginReqPlsDataModeMan := (#StartCmdPlsMan AND #DataModeMan);

   #IO_VIDS.GetSpecData.BeginReq := #BeginReqPlsDataModeAuto OR #BeginReqPlsDataModeMan;

   IF  #IO_VIDS.GetSpecData.BeginReq THEN
       #Status := 0;
       #TagIDMem := #I_TagID;
       #BodyIDMem := #I_BodyID;
       #CarrierIDMem := #I_CarrierID;
       #MixNrMem := #I_MixNr;
       #PopIDMem := #I_PopID;
       #PopIDSuffixMem := #I_PopIDSuffix;
       #PopTypeMem := #I_PopType;
   END_IF;

   (******************************************************************************)
   (* OkBegin / Begin / Running                                                  *)
   (******************************************************************************)
   //OkBegin
   IF  #IO_VIDS.GetSpecData.OkBegin THEN
       #DataValid := False;
       #DataNotValid := False;
       #IO_VIDS.VEMData.FunctionCode := 0; //>>> MOET "0" ZIJN >>> DECODE YOUR DATA HERE!
       #IO_VIDS.VEMData.CommandCode := #C_Command; //>>> DECODE YOUR DATA HERE!
       #IO_VIDS.VEMData.Identification:= #TagIDMem; //>>> DECODE YOUR DATA HERE!
       #IO_VIDS.VEMData.BodyID:= #BodyIDMem; //>>> DECODE YOUR DATA HERE!
       #IO_VIDS.VEMData.CarrierID := #CarrierIDMem; //>>> DECODE YOUR DATA HERE!
       #IO_VIDS.VEMData.MixNumber := #MixNrMem; //>>> DECODE YOUR DATA HERE!
       #IO_VIDS.VEMData.PopID := #PopIDMem; //>>> DECODE YOUR DATA HERE!
       #IO_VIDS.VEMData.PopIDSuffix := #PopIDSuffixMem; //>>> DECODE YOUR DATA HERE!
       #IO_VIDS.VEMData.PopType := #PopTypeMem; //>>> DECODE YOUR DATA HERE!
   END_IF;

   //Begin
   #IO_VIDS.GetSpecData.Begin := #IO_VIDS.GetSpecData.OkBegin;

   //Running
   IF #IO_VIDS.GetSpecData.Running THEN
       #Status := #IO_VIDS.GetSpecData.Status;
   END_IF;

   (******************************************************************************)
   (* Finish                                                                     *)
   (******************************************************************************)
   IF #IO_VIDS.GetSpecData.Finished THEN
       #Status := #IO_VIDS.GetSpecData.Status;

       IF #Status = 1 THEN
           #BodyType1 := #IO_VIDS.VEMData.BodyType1; //>>> DECODE YOUR DATA HERE! 
           #VemData := #IO_VIDS.VEMData; //>>> DECODE YOUR DATA HERE! 
           #DataValid := TRUE;
       ELSE
               #DataNotValid := TRUE;
       END_IF;

   END_IF;

   (******************************************************************************************************************************)
   (* EINDE COMMUNICATION WITH IT                                                                                                *)
   (******************************************************************************************************************************)

   (******************************************************************************)
   (* Clear data                                                                 *)
   (******************************************************************************)
   IF #IO_VIDS.GetSpecData.BeginReq OR #DataModeChanged OR NOT #IO_VIDS.PartPres THEN
       #DataValid := False;
       #DataNotValid := False;
       #Status := 0;
       #BodyType1 := 0;//>>> DECODE YOUR DATA HERE! 
       #VemData := #VemDataEmty;//>>> DECODE YOUR DATA HERE! 

   END_IF;

   IF NOT #IO_VIDS.PartPres THEN
       #TagIDMem := 0;//>>> DECODE YOUR DATA HERE!
       #BodyIDMem := 0;//>>> DECODE YOUR DATA HERE!
       #CarrierIDMem := 0;//>>> DECODE YOUR DATA HERE!
       #MixNrMem := 0;//>>> DECODE YOUR DATA HERE!
       #PopIDMem := 0;//>>> DECODE YOUR DATA HERE!
       #PopIDSuffixMem := ' ';//>>> DECODE YOUR DATA HERE!
       #PopTypeMem := 0;//>>> DECODE YOUR DATA HERE!
   END_IF;

   (******************************************************************************)
   (* Alarm = status <0                                                          *)
   (******************************************************************************)
   IF #Status < 0 THEN
       #Alarm := TRUE;
   ELSE
       #Alarm := false;
   END_IF;

   "LAlarmSummary"(I_AlarmA := FALSE,
                   I_AlarmB := FALSE,
                   I_AlarmC := #Alarm,
                   I_AlarmD := FALSE,
                   I_AlarmABCondition := FALSE,
                   IO_Alarm := #IO_Alarm,
                   C_UpperLevelHW := "FALSE",
                   C_UpperLevelSafety := "FALSE",
                   C_Safety := "FALSE",
                   C_Mechanic := "FALSE",
                   C_Transport := "FALSE",
                   C_Feature1 := "FALSE",
                   C_Feature2 := "FALSE",
                   C_Feature3 := "FALSE");

   (******************************************************************************)
   (* Calculation BodyCargoStatus OK - NOK                                       *)
   (******************************************************************************)

   IF #VemData.BodyCargoStatus.%X0 = true THEN
       #BodyCargoStatusOk := TRUE;
   ELSE
       #BodyCargoStatusOk := FALSE;
   END_IF;

   IF #VemData.BodyCargoStatus.%X1 = true THEN
       #BodyCargoStatusNok := TRUE;
   ELSE
       #BodyCargoStatusNok := FALSE;
   END_IF;

   (******************************************************************************)
   (* Outputs                                                                    *)
   (******************************************************************************)
   #O_DataModeAuto := #DataModeAuto;
   #O_DataModeMan := #DataModeMan;
   #O_DataValid := #DataValid;
   #O_DataNotValid := #DataNotValid;
   #O_Alarm := #Alarm;
   #O_Status := #Status;
   #O_Busy := #IO_VIDS.GetSpecData.Running;
   #O_VemData := #VemData;                         //>>> DECODE YOUR DATA HERE!
   #O_BodyCargoStatusOk := #BodyCargoStatusOk;     //>>> DECODE YOUR DATA HERE!
   #O_BodyCargoStatusNok := #BodyCargoStatusNok;   //>>> DECODE YOUR DATA HERE!

   (******************************************************************************************************************************)
   (* Animations                                                                                                                 *)
   (******************************************************************************************************************************)

   (******************************************************************************)
   (* Status To HMI word                                                         *)
   (******************************************************************************)
   "LBitToDword"(I_0:=#IO_VIDS.PartPres,
                 I_1:=#DataValid,
                 I_2:=#DataNotValid,
                 I_3:=#Alarm,
                 I_4:=#I_Start,
                 I_5:=#H_LVIDSQualityRequest.H_selDataMode = 3,
                 I_6:=FALSE,
                 I_7:=FALSE,
                 I_8:=FALSE,
                 I_9:=FALSE,
                 I_10:=FALSE,
                 I_11:=FALSE,
                 I_12:=FALSE,
                 I_13:=FALSE,
                 I_14:=FALSE,
                 I_15:=FALSE,
                 I_16:=FALSE,
                 I_17:=FALSE,
                 I_18:=FALSE,
                 I_19:=FALSE,
                 I_20:=FALSE,
                 I_21:=FALSE,
                 I_22:=FALSE,
                 I_23:=FALSE,
                 I_24:=FALSE,
                 I_25:=FALSE,
                 I_26:=FALSE,
                 I_27:=FALSE,
                 I_28:=FALSE,
                 I_29:=FALSE,
                 I_30:=FALSE,
                 I_31:=FALSE,
                 O_DWord=>#H_LVIDSQualityRequest.H_Anim);

   (******************************************************************************)
   (* Status To HMI word - IAnim                                                 *)
   (******************************************************************************)
   //*** Machine #Status - Indication *** TO HMI - Icon animation
   "LIAnimDWord"(I_SetPos:=FALSE,
                 I_ResetPos:=FALSE,
                 I_Active:=#Status=2,
                 I_Visible:=FALSE,
                 I_OutOfUse:=FALSE,
                 I_IntlkSet:=FALSE,
                 I_IntlkReset:=FALSE,
                 I_IntlkSetAlm:=FALSE,
                 I_IntlkResetAlm:=FALSE,
                 I_ManualMode:=FALSE,
                 I_FncSelInHMI:=FALSE,
                 I_AnySelected:=FALSE,
                 I_AlarmA:=FALSE,
                 I_AlarmB:=FALSE,
                 I_AlarmC:=#DataNotValid,
                 I_AlarmD:=FALSE,
                 I_SafetyOk:=FALSE,
                 I_Service:=TRUE,
                 I_Spare1:=FALSE,
                 I_Spare2:=FALSE,
                 I_Spare3:=FALSE,
                 I_Spare4:=FALSE,
                 I_Spare5:=FALSE,
                 I_Spare6:=FALSE,
                 I_Spare7:=FALSE,
                 I_Spare8:=FALSE,
                 I_Spare9:=FALSE,
                 I_Spare10:=FALSE,
                 I_Spare11:=FALSE,
                 I_Spare12:=FALSE,
                 I_Spare13:=FALSE,
                 I_Spare14:=FALSE,
                 H_IAnim=>#H_HMI.H_IAnim);

   (******************************************************************************)
   (* Copy Txt info to HMI                                                       *)
   (******************************************************************************)
   #H_LVIDSQualityRequest.H_txtStatusIT := #Status;
   #H_LVIDSQualityRequest.H_txtBodyCargoStatus := #VemData.BodyCargoStatus;
   #H_LVIDSQualityRequest.H_txtRouting := #VemData.Routing;
   #H_LVIDSQualityRequest.H_txtPopType := #VemData.PopType;
   #H_LVIDSQualityRequest.H_txtPopId := #VemData.PopID;
   #H_LVIDSQualityRequest.H_txtPopIdSuffix := #VemData.PopIDSuffix;

   #H_LVIDSQualityRequest.H_txtInTagID := #TagIDMem;
   #H_LVIDSQualityRequest.H_txtInBodyID := #BodyIDMem;
   #H_LVIDSQualityRequest.H_txtInCarrierID := #CarrierIDMem;
   #H_LVIDSQualityRequest.H_txtInMixNr := #MixNrMem;
   #H_LVIDSQualityRequest.H_txtInPopId := #PopIDMem;
   #H_LVIDSQualityRequest.H_txtInPopIdSuffix := #PopIDSuffixMem;
   #H_LVIDSQualityRequest.H_txtInPopType := #PopTypeMem;

   #H_LVIDSQualityRequest.H_txtCommandCodeRcvd := #IO_VIDS.CmdCodeRcvd;
   #H_LVIDSQualityRequest.H_txtCommandCodeSent := #IO_VIDS.CmdCodeSent;

   (******************************************************************************)
   (* Animation BUTTONS                                                          *)
   (******************************************************************************)
   //Data mode manual - <Confirm> button
   IF #I_ManualModeVisible AND #DataModeMan THEN
       #H_btnConfirmDataModeManVisible := #VISIBLE;
       #H_btnConfirmDataModeManEnable := #ENABLE;
   ELSE
       #H_btnConfirmDataModeManVisible := #OFF;
       #H_btnConfirmDataModeManEnable := #OFF;
   END_IF;

   #H_LVIDSQualityRequest.H_btnConfirmDataModeManAnim := #H_btnConfirmDataModeManEnable OR #H_btnConfirmDataModeManVisible;
END_FUNCTION_BLOCK

FUNCTION_BLOCK "L2StopPos"   // FB1310, FBD
TITLE = L2StopPos
{ S7_Optimized_Access := 'TRUE' }
AUTHOR : VCC
FAMILY : Actuator
VERSION : 0.1
// =============================================================================
// This module will be used for a two Position movements.
// It will take care of the Alarms and of the Detections.
// =============================================================================
// stored: AutoNumber false, IsIECCheckEnabled false, IsRetainMemResEnabled false, MemoryReserve 100, SetENOAutomatically False, UDAEnableTagReadback false
   VAR_INPUT
      I_DetSet { ExternalAccessible := 'False'; ExternalVisible := 'False'; ExternalWritable := 'False'} : Bool;   // Set detection signal / Set Detection signal
      I_DetRes { ExternalAccessible := 'False'; ExternalVisible := 'False'; ExternalWritable := 'False'} : Bool;   // Reset detection signal / Reset Detection signal
      I_CmdSet { ExternalAccessible := 'False'; ExternalVisible := 'False'; ExternalWritable := 'False'} : Bool;   // function set command / Function set command
      I_CmdRes { ExternalAccessible := 'False'; ExternalVisible := 'False'; ExternalWritable := 'False'} : Bool;   // Function reset command / Function Reset command
      I_RunSet { ExternalAccessible := 'False'; ExternalVisible := 'False'; ExternalWritable := 'False'} : Bool;   // Memory that the Set function is busy
      I_RunRes { ExternalAccessible := 'False'; ExternalVisible := 'False'; ExternalWritable := 'False'} : Bool;   // Memory that the Reset function is busy
      I_SetIntlkOK { ExternalAccessible := 'False'; ExternalVisible := 'False'; ExternalWritable := 'False'} : Bool := TRUE;   // Set Interlock
      I_ResIntlkOK { ExternalAccessible := 'False'; ExternalVisible := 'False'; ExternalWritable := 'False'} : Bool := TRUE;   // Reset Interlock
      I_SafetyOk { ExternalAccessible := 'False'; ExternalVisible := 'False'; ExternalWritable := 'False'} : Bool;   // Safety Ok
      I_AlarmResetPB { ExternalAccessible := 'False'; ExternalVisible := 'False'; ExternalWritable := 'False'} : Bool := TRUE;   // alarm reset Push Button is activated / Alarm Reset Push Button is Activated
      C_KeepPosition { ExternalAccessible := 'False'; ExternalVisible := 'False'; ExternalWritable := 'False'} : Bool;   // If true, the last position shall be kept ON and checked / If true, the last Position shall be kept ON and checked
      C_EnAlmDet { ExternalAccessible := 'False'; ExternalVisible := 'False'; ExternalWritable := 'False'} : Bool;   // Enable alarm / Enable Alarm
      C_AlarmResetUsed { ExternalAccessible := 'False'; ExternalVisible := 'False'; ExternalWritable := 'False'} : Bool;   // If true, the alarms will be stored untill reseted / If true, the Alarms will be stored untill Reseted
      C_EnAlmOvertime { ExternalAccessible := 'False'; ExternalVisible := 'False'; ExternalWritable := 'False'} : Bool := TRUE;   // Enable Overtime Alarm
      C_ManualClampCmdSet { ExternalAccessible := 'False'; ExternalVisible := 'False'; ExternalWritable := 'False'} : Bool;   // Manual Clamp Set
      C_ManualClampCmdRes { ExternalAccessible := 'False'; ExternalVisible := 'False'; ExternalWritable := 'False'} : Bool;   // Manual Clamp Reset
      C_RunTimeMaxSetWarn { ExternalAccessible := 'False'; ExternalVisible := 'False'; ExternalWritable := 'False'} : DInt;   // Maximum Time (ms) that the function may run (create overtime) / Maximum Time (ms) that the function may run (create Overtime)
      C_RunTimeMaxSetAlm { ExternalAccessible := 'False'; ExternalVisible := 'False'; ExternalWritable := 'False'} : DInt;   // Maximum Time (ms) that the function may run (create overtime) / Maximum Time (ms) that the function may run (create Overtime)
      C_RunTimeMaxResWarn { ExternalAccessible := 'False'; ExternalVisible := 'False'; ExternalWritable := 'False'} : DInt;   // Maximum Time (ms) that the function may run (create overtime) / Maximum Time (ms) that the function may run (create Overtime)
      C_RunTimeMaxResAlm { ExternalAccessible := 'False'; ExternalVisible := 'False'; ExternalWritable := 'False'} : DInt;   // Maximum Time (ms) that the function may run (create overtime) / Maximum Time (ms) that the function may run (create Overtime)
      C_TimeAlmFilt { ExternalAccessible := 'False'; ExternalVisible := 'False'; ExternalWritable := 'False'} : DInt := L#2000;   // timer before any actuator alarm will be active (welding..) / timer before any actuator Alarm will be active (welding..)
      C_AlarmSeverityAB { ExternalAccessible := 'False'; ExternalVisible := 'False'; ExternalWritable := 'False'} : Bool;   // Alarm severity
      C_RunTimeCalculated { ExternalAccessible := 'False'; ExternalVisible := 'False'; ExternalWritable := 'False'} : Bool;   // Maximum Time (ms) that the function may run (create Overtime) is calculated
   END_VAR
   VAR_OUTPUT
      O_SetPos { ExternalAccessible := 'False'; ExternalVisible := 'False'; ExternalWritable := 'False'} : Bool;   // Actuator is in set position / Actuator is in set Position
      O_ResPos { ExternalAccessible := 'False'; ExternalVisible := 'False'; ExternalWritable := 'False'} : Bool;   // Actuator is in reset position / Actuator is in Reset Position
      O_KeepPosSetAlm { ExternalAccessible := 'False'; ExternalVisible := 'False'; ExternalWritable := 'False'} : Bool;   // Detection Set alarm / Detection Set Alarm
      O_KeepPosResAlm { ExternalAccessible := 'False'; ExternalVisible := 'False'; ExternalWritable := 'False'} : Bool;   // Detection Reset alarm / Detection Reset Alarm
      O_TwoDetAlm { ExternalAccessible := 'False'; ExternalVisible := 'False'; ExternalWritable := 'False'} : Bool;   // Fault condition Both detections ON at the same time
      O_OvtSetWarn { ExternalAccessible := 'False'; ExternalVisible := 'False'; ExternalWritable := 'False'} : Bool;   // Warning Overtime Set
      O_OvtResWarn { ExternalAccessible := 'False'; ExternalVisible := 'False'; ExternalWritable := 'False'} : Bool;   // Warning Overtime Reset
      O_OvtSetAlm { ExternalAccessible := 'False'; ExternalVisible := 'False'; ExternalWritable := 'False'} : Bool;   // Alarm Overtime Set
      O_OvtResAlm { ExternalAccessible := 'False'; ExternalVisible := 'False'; ExternalWritable := 'False'} : Bool;   // Alarm Overtime Reset
      O_ConfigCalibrationAlm { ExternalAccessible := 'False'; ExternalVisible := 'False'; ExternalWritable := 'False'} : Bool;   // Alarm Config/Calibration
      O_CalibrationWarn { ExternalAccessible := 'False'; ExternalVisible := 'False'; ExternalWritable := 'False'} : Bool;   // Warning Calibration
      O_AlarmABCondition { ExternalAccessible := 'False'; ExternalVisible := 'False'; ExternalWritable := 'False'} : Bool;   // Alarm AB condition / Alarm AB Condition
      H_IAnim { ExternalAccessible := 'False'; ExternalVisible := 'False'; ExternalWritable := 'False'} : DWord;   // Animation color of icon
   END_VAR
   VAR_IN_OUT
      IO_Modes : "Modes";   // Modes
      H_2StopPos : "H_2StopPos";   // Animation
   END_VAR
   VAR
      AlarmReset { ExternalAccessible := 'False'; ExternalVisible := 'False'; ExternalWritable := 'False'} : Bool;   // Alarm Reset Memory
      SetPosReq { ExternalAccessible := 'False'; ExternalVisible := 'False'; ExternalWritable := 'False'} : Bool;   // Memorisation of the last set movement
      ResPosReq { ExternalAccessible := 'False'; ExternalVisible := 'False'; ExternalWritable := 'False'} : Bool;   // Memorisation of the last reset movement / Memorisation of the last Reset movement
      KeepSetPosOn { ExternalAccessible := 'False'; ExternalVisible := 'False'; ExternalWritable := 'False'} : Bool;   // Check that Set detection is keept on / Check that Set Detection is keept on
      KeepResPosOn { ExternalAccessible := 'False'; ExternalVisible := 'False'; ExternalWritable := 'False'} : Bool;   // Check that Set detection is keept on / Check that Set Detection is keept on
      KeepPosSetStartTimer { ExternalAccessible := 'False'; ExternalVisible := 'False'; ExternalWritable := 'False'} : Bool;   // Detection Set request to start timer / Detection Set Request to start timer
      KeepPosResStartTimer { ExternalAccessible := 'False'; ExternalVisible := 'False'; ExternalWritable := 'False'} : Bool;   // Detection Reset request to start timer / Detection Reset Request to start timer
      TwoDetStartTimer { ExternalAccessible := 'False'; ExternalVisible := 'False'; ExternalWritable := 'False'} : Bool;   // Both detections ON at the same time request to start timer / Both Detections ON at the same time Request to start timer
      AlarmFilterStart { ExternalAccessible := 'False'; ExternalVisible := 'False'; ExternalWritable := 'False'} : Bool;   // Alarm filter must be started
      OvtSetWarnResult { ExternalAccessible := 'False'; ExternalVisible := 'False'; ExternalWritable := 'False'} : Bool;   // Overtime set warning result
      OvtResWarnResult { ExternalAccessible := 'False'; ExternalVisible := 'False'; ExternalWritable := 'False'} : Bool;   // Overtime reset warning result / Overtime Reset warning result
      OvtSetAlmResult { ExternalAccessible := 'False'; ExternalVisible := 'False'; ExternalWritable := 'False'} : Bool;   // Overtime set alarm result / Overtime set Alarm result
      OvtResAlmResult { ExternalAccessible := 'False'; ExternalVisible := 'False'; ExternalWritable := 'False'} : Bool;   // Overtime reset alarm result / Overtime Reset Alarm result
      AlmFilterResult { ExternalAccessible := 'False'; ExternalVisible := 'False'; ExternalWritable := 'False'} : Bool;   // Alarm filter result
      TwoDetAlm { ExternalAccessible := 'False'; ExternalVisible := 'False'; ExternalWritable := 'False'} : Bool;   // Two detection alarm / Set Reset Activated Simultaneously / Set Reset Påverkade Samtidigt
      KeepPosResAlm { ExternalAccessible := 'False'; ExternalVisible := 'False'; ExternalWritable := 'False'} : Bool;   // Keep position Reset alarm / Position Supervision Reset Position / Positionsövervakning Reset Läge
      KeepPosSetAlm { ExternalAccessible := 'False'; ExternalVisible := 'False'; ExternalWritable := 'False'} : Bool;   // Keep position Set alarm / Alarm Keep Position Set Position / Larm Positionsövervakning Set Läge
      OvtResAlm { ExternalAccessible := 'False'; ExternalVisible := 'False'; ExternalWritable := 'False'} : Bool;   // Overtime Reset alarm / Overtime Reset Alarm
      OvtSetAlm { ExternalAccessible := 'False'; ExternalVisible := 'False'; ExternalWritable := 'False'} : Bool;   // Overtime Set alarm / Timeout Set / Tidsövervakning Set
      OvtResWarn { ExternalAccessible := 'False'; ExternalVisible := 'False'; ExternalWritable := 'False'} : Bool;   // Overtime Reset warning
      OvtSetWarn { ExternalAccessible := 'False'; ExternalVisible := 'False'; ExternalWritable := 'False'} : Bool;   // Overtime Set warning
      ConfigCalibrationAlm { ExternalAccessible := 'False'; ExternalVisible := 'False'; ExternalWritable := 'False'} : Bool;   // Config/Calibration Alarm
      CalibrationWarn { ExternalAccessible := 'False'; ExternalVisible := 'False'; ExternalWritable := 'False'} : Bool;   // Warning Calibration
      SetPos { ExternalAccessible := 'False'; ExternalVisible := 'False'; ExternalWritable := 'False'} : Bool;   // Set position / Set Position
      ResPos { ExternalAccessible := 'False'; ExternalVisible := 'False'; ExternalWritable := 'False'} : Bool;   // Reset position / Reset Position
      KeepPosResAlmCond { ExternalAccessible := 'False'; ExternalVisible := 'False'; ExternalWritable := 'False'} : Bool;   // Keep position reset alarm condition / Keep Position Reset Alarm condition
      KeepPosSetAlmCond { ExternalAccessible := 'False'; ExternalVisible := 'False'; ExternalWritable := 'False'} : Bool;   // Keep position set alarm condition / Keep Position Set Alarm condition
      TwoDetAlmCond { ExternalAccessible := 'False'; ExternalVisible := 'False'; ExternalWritable := 'False'} : Bool;   // Two detector alarm condition / Two detector Alarm condition
      OvtResAlmCond { ExternalAccessible := 'False'; ExternalVisible := 'False'; ExternalWritable := 'False'} : Bool;   // Overtime reset alarm condition / Overtime Reset Alarm condition
      OvtSetAlmCond { ExternalAccessible := 'False'; ExternalVisible := 'False'; ExternalWritable := 'False'} : Bool;   // Overtime set alarm condition / Overtime set Alarm condition
      RunSet { ExternalAccessible := 'False'; ExternalVisible := 'False'; ExternalWritable := 'False'} : Bool;   // Memory that the Set function is busy
      RunRes { ExternalAccessible := 'False'; ExternalVisible := 'False'; ExternalWritable := 'False'} : Bool;   // Memory that the Reset function is busy
      Edge { ExternalAccessible := 'False'; ExternalVisible := 'False'; ExternalWritable := 'False'} : Array[1..8] of Bool;   // Edge
      AlarmTimer { ExternalAccessible := 'False'; ExternalVisible := 'False'; ExternalWritable := 'False'} : "LTimer";   // FB
      OvtSetWarnTimer { ExternalAccessible := 'False'; ExternalVisible := 'False'; ExternalWritable := 'False'} : "LTimer";   // FB
      OvtResWarnTimer { ExternalAccessible := 'False'; ExternalVisible := 'False'; ExternalWritable := 'False'} : "LTimer";   // FB
      OvtSetAlmTimer { ExternalAccessible := 'False'; ExternalVisible := 'False'; ExternalWritable := 'False'} : "LTimer";   // FB
      OvtResAlmTimer { ExternalAccessible := 'False'; ExternalVisible := 'False'; ExternalWritable := 'False'} : "LTimer";   // FB
   END_VAR
   VAR RETAIN
      OvtWarnSet { ExternalAccessible := 'False'; ExternalVisible := 'False'; ExternalWritable := 'False'} : DInt;   // Alarm Value
      OvtWarnRes { ExternalAccessible := 'False'; ExternalVisible := 'False'; ExternalWritable := 'False'} : DInt;   // Alarm Value
      OvtAlarmSet { ExternalAccessible := 'False'; ExternalVisible := 'False'; ExternalWritable := 'False'} : DInt;   // Alarm Value
      OvtAlarmRes { ExternalAccessible := 'False'; ExternalVisible := 'False'; ExternalWritable := 'False'} : DInt;   // Alarm Value
      CalibratedSet { ExternalAccessible := 'False'; ExternalVisible := 'False'; ExternalWritable := 'False'} : Bool;   // Calibrated Set
      CalibratedRes { ExternalAccessible := 'False'; ExternalVisible := 'False'; ExternalWritable := 'False'} : Bool;   // Calibrated Reset
   END_VAR
   VAR
      AlarmTimeWithConfig { ExternalAccessible := 'False'; ExternalVisible := 'False'; ExternalWritable := 'False'} : Bool;
      AlarmTimeWithCalibration { ExternalAccessible := 'False'; ExternalVisible := 'False'; ExternalWritable := 'False'} : Bool;
      AlarmTimeWithCalculation { ExternalAccessible := 'False'; ExternalVisible := 'False'; ExternalWritable := 'False'} : Bool;
      AlmFilterTimerValue { ExternalAccessible := 'False'; ExternalVisible := 'False'; ExternalWritable := 'False'} : DInt;
   END_VAR
   VAR_TEMP
      H_CalibrateSet : Bool;   // HMI Function
      H_CalibrateReset : Bool;   // HMI Function
      TempReal : Real;
   END_VAR
   VAR_TEMP   // added for the SCL form of the ladder/FBD networks
      _w1 : Bool;
      _w2 : Bool;
      _w3 : Bool;
      _w4 : Bool;
   END_VAR
BEGIN

REGION Network 1: **** 1 - Inputs **** HMI Commands
   // Extract the Commands from HMIRobCmd / Extract the Commands from HMI
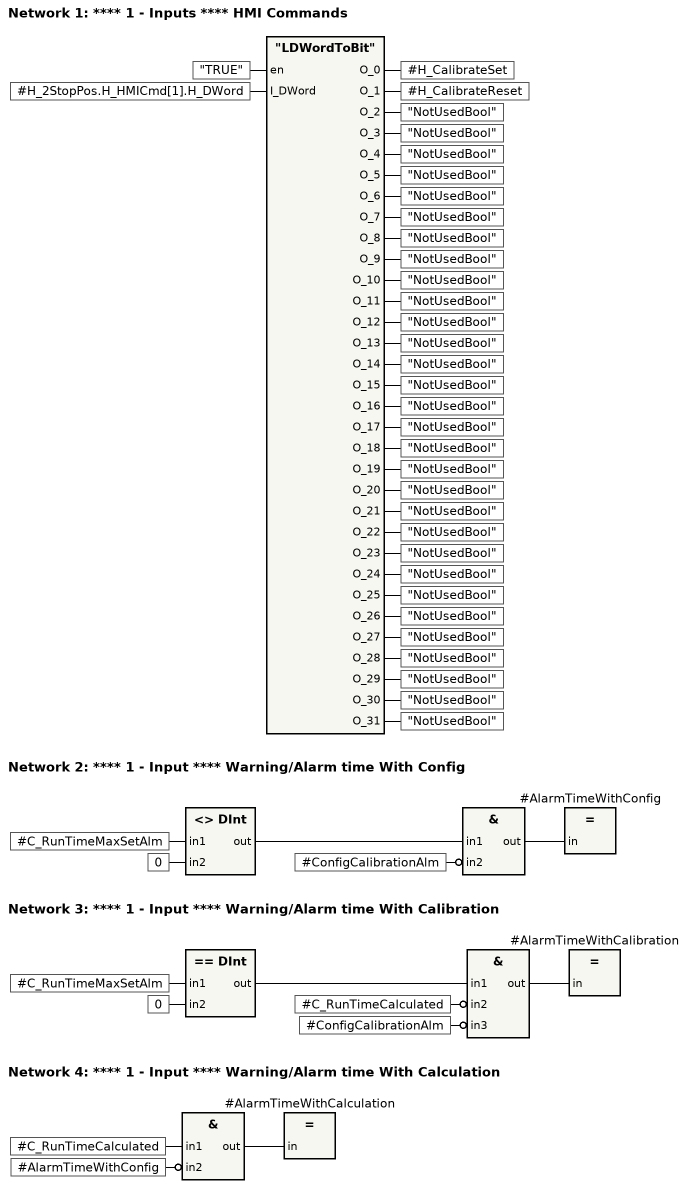
   IF "TRUE" THEN
       "LDWordToBit"(I_DWord := #H_2StopPos.H_HMICmd[1].H_DWord,
                     O_0 => #H_CalibrateSet,
                     O_1 => #H_CalibrateReset,
                     O_2 => "NotUsedBool",
                     O_3 => "NotUsedBool",
                     O_4 => "NotUsedBool",
                     O_5 => "NotUsedBool",
                     O_6 => "NotUsedBool",
                     O_7 => "NotUsedBool",
                     O_8 => "NotUsedBool",
                     O_9 => "NotUsedBool",
                     O_10 => "NotUsedBool",
                     O_11 => "NotUsedBool",
                     O_12 => "NotUsedBool",
                     O_13 => "NotUsedBool",
                     O_14 => "NotUsedBool",
                     O_15 => "NotUsedBool",
                     O_16 => "NotUsedBool",
                     O_17 => "NotUsedBool",
                     O_18 => "NotUsedBool",
                     O_19 => "NotUsedBool",
                     O_20 => "NotUsedBool",
                     O_21 => "NotUsedBool",
                     O_22 => "NotUsedBool",
                     O_23 => "NotUsedBool",
                     O_24 => "NotUsedBool",
                     O_25 => "NotUsedBool",
                     O_26 => "NotUsedBool",
                     O_27 => "NotUsedBool",
                     O_28 => "NotUsedBool",
                     O_29 => "NotUsedBool",
                     O_30 => "NotUsedBool",
                     O_31 => "NotUsedBool");
   END_IF;
END_REGION

REGION Network 2: **** 1 - Input **** Warning/Alarm time With Config
   #AlarmTimeWithConfig := (#C_RunTimeMaxSetAlm <> 0) AND NOT #ConfigCalibrationAlm;
END_REGION

REGION Network 3: **** 1 - Input **** Warning/Alarm time With Calibration
   #AlarmTimeWithCalibration := (#C_RunTimeMaxSetAlm = 0) AND NOT #C_RunTimeCalculated AND NOT #ConfigCalibrationAlm;
END_REGION

REGION Network 4: **** 1 - Input **** Warning/Alarm time With Calculation
   #AlarmTimeWithCalculation := #C_RunTimeCalculated AND NOT #AlarmTimeWithConfig;
END_REGION

REGION Network 5: Calibrated Set / **** 1 - Input **** Ovt Values / **** 1 - Inputs **** Ovt Values
   // Ovt Values
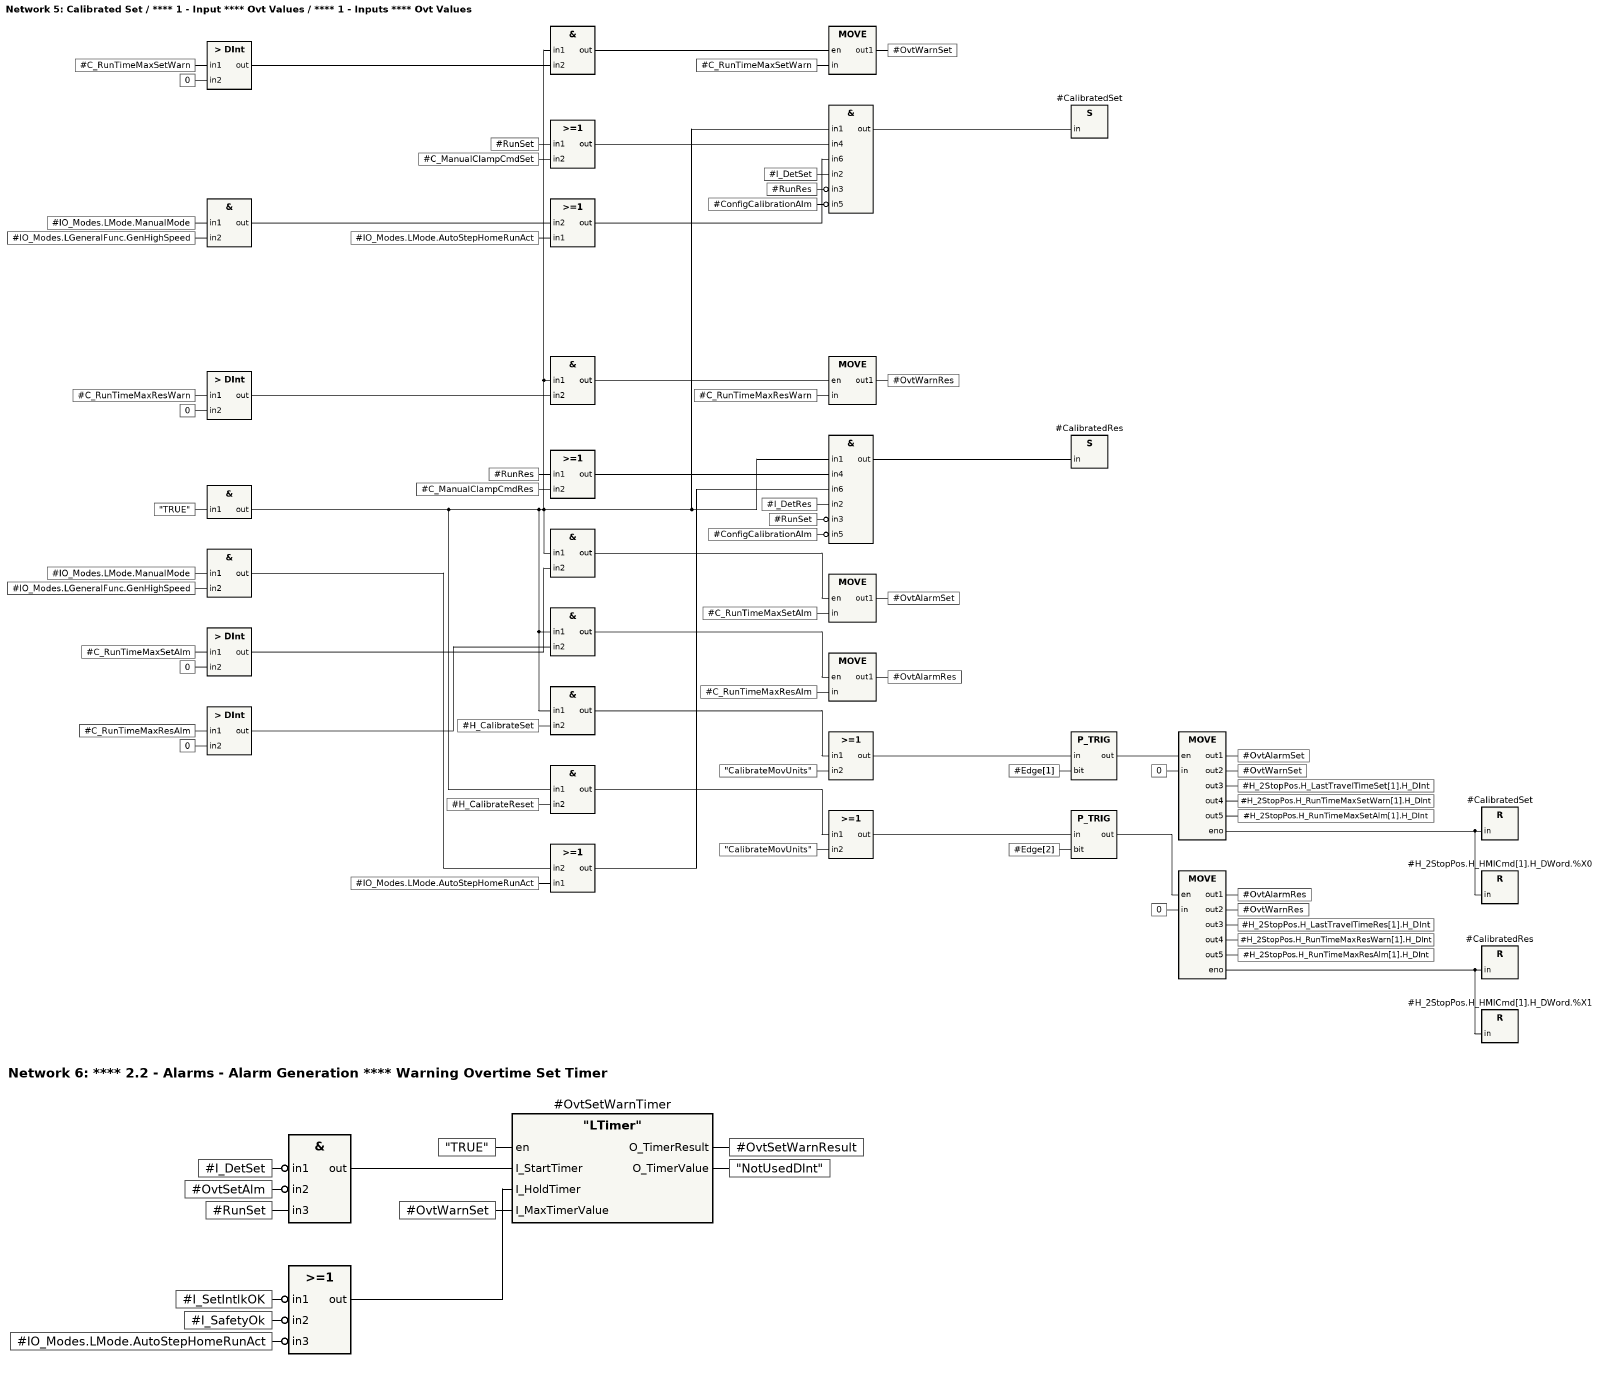
   // ENO of a box is taken as its EN; it also drops when the box reports an error
   IF "TRUE" AND (#C_RunTimeMaxSetWarn > 0) THEN #OvtWarnSet := #C_RunTimeMaxSetWarn; END_IF;
   IF "TRUE" AND (#C_RunTimeMaxResWarn > 0) THEN #OvtWarnRes := #C_RunTimeMaxResWarn; END_IF;
   IF "TRUE" AND (#C_RunTimeMaxSetAlm > 0) THEN #OvtAlarmSet := #C_RunTimeMaxSetAlm; END_IF;
   IF "TRUE" AND (#C_RunTimeMaxResAlm > 0) THEN #OvtAlarmRes := #C_RunTimeMaxResAlm; END_IF;
   IF "TRUE" AND (#RunSet OR #C_ManualClampCmdSet) AND ((#IO_Modes.LMode.ManualMode AND #IO_Modes.LGeneralFunc.GenHighSpeed) OR #IO_Modes.LMode.AutoStepHomeRunAct) AND #I_DetSet AND NOT #RunRes AND NOT #ConfigCalibrationAlm THEN
       #CalibratedSet := TRUE;
   END_IF;
   IF "TRUE" AND (#RunRes OR #C_ManualClampCmdRes) AND ((#IO_Modes.LMode.ManualMode AND #IO_Modes.LGeneralFunc.GenHighSpeed) OR #IO_Modes.LMode.AutoStepHomeRunAct) AND #I_DetRes AND NOT #RunSet AND NOT #ConfigCalibrationAlm THEN
       #CalibratedRes := TRUE;
   END_IF;
   #_w1 := ("TRUE" AND #H_CalibrateSet) OR "CalibrateMovUnits";
   #_w2 := #_w1 AND NOT #Edge[1];   // rising edge
   #Edge[1] := #_w1;
   IF #_w2 THEN
       #OvtAlarmSet := 0;
       #OvtWarnSet := 0;
       #H_2StopPos.H_LastTravelTimeSet[1].H_DInt := 0;
       #H_2StopPos.H_RunTimeMaxSetWarn[1].H_DInt := 0;
       #H_2StopPos.H_RunTimeMaxSetAlm[1].H_DInt := 0;
       #CalibratedSet := FALSE;
       #H_2StopPos.H_HMICmd[1].H_DWord.%X0 := FALSE;
   END_IF;
   #_w3 := ("TRUE" AND #H_CalibrateReset) OR "CalibrateMovUnits";
   #_w4 := #_w3 AND NOT #Edge[2];   // rising edge
   #Edge[2] := #_w3;
   IF #_w4 THEN
       #OvtAlarmRes := 0;
       #OvtWarnRes := 0;
       #H_2StopPos.H_LastTravelTimeRes[1].H_DInt := 0;
       #H_2StopPos.H_RunTimeMaxResWarn[1].H_DInt := 0;
       #H_2StopPos.H_RunTimeMaxResAlm[1].H_DInt := 0;
       #CalibratedRes := FALSE;
       #H_2StopPos.H_HMICmd[1].H_DWord.%X1 := FALSE;
   END_IF;
END_REGION

REGION Network 6: **** 2.2 - Alarms - Alarm Generation **** Warning Overtime Set Timer
   // Warning Overtime Set Timer
   IF "TRUE" THEN
       #OvtSetWarnTimer(I_StartTimer := NOT #I_DetSet AND NOT #OvtSetAlm AND #RunSet,   // "LTimer"
                        I_HoldTimer := NOT #I_SetIntlkOK OR NOT #I_SafetyOk OR NOT #IO_Modes.LMode.AutoStepHomeRunAct,
                        I_MaxTimerValue := #OvtWarnSet,
                        O_TimerResult => #OvtSetWarnResult,
                        O_TimerValue => "NotUsedDInt");
   END_IF;
END_REGION

REGION Network 7: **** 2.2 - Alarms - Alarm Generation **** Warning Overtime Set Memorisation
   // Warning Overtime Set Memorisation
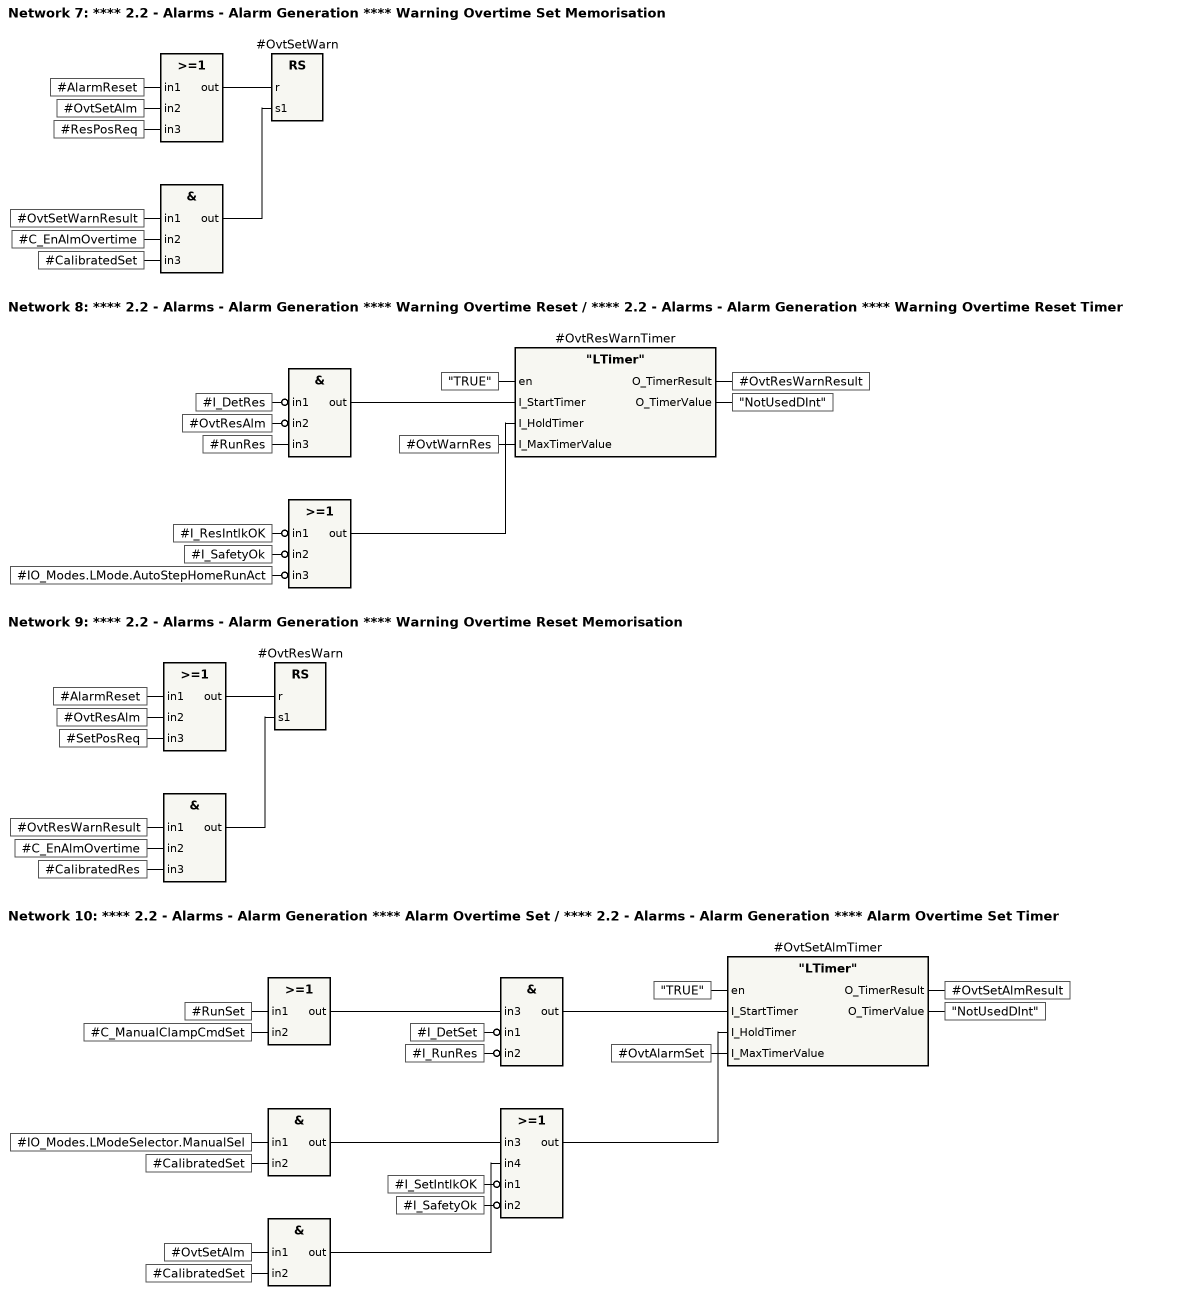
   IF #AlarmReset OR #OvtSetAlm OR #ResPosReq THEN
       #OvtSetWarn := FALSE;   // RS flip-flop
   END_IF;
   IF #OvtSetWarnResult AND #C_EnAlmOvertime AND #CalibratedSet THEN #OvtSetWarn := TRUE; END_IF;
END_REGION

REGION Network 8: **** 2.2 - Alarms - Alarm Generation **** Warning Overtime Reset / **** 2.2 - Alarms - Alarm Generation **** Warning Overtime Reset Timer
   // Warning Overtime Reset
   IF "TRUE" THEN
       #OvtResWarnTimer(I_StartTimer := NOT #I_DetRes AND NOT #OvtResAlm AND #RunRes,   // "LTimer"
                        I_HoldTimer := NOT #I_ResIntlkOK OR NOT #I_SafetyOk OR NOT #IO_Modes.LMode.AutoStepHomeRunAct,
                        I_MaxTimerValue := #OvtWarnRes,
                        O_TimerResult => #OvtResWarnResult,
                        O_TimerValue => "NotUsedDInt");
   END_IF;
END_REGION

REGION Network 9: **** 2.2 - Alarms - Alarm Generation **** Warning Overtime Reset Memorisation
   // Warning Overtime Reset  Memorisation
   IF #AlarmReset OR #OvtResAlm OR #SetPosReq THEN
       #OvtResWarn := FALSE;   // RS flip-flop
   END_IF;
   IF #OvtResWarnResult AND #C_EnAlmOvertime AND #CalibratedRes THEN #OvtResWarn := TRUE; END_IF;
END_REGION

REGION Network 10: **** 2.2 - Alarms - Alarm Generation **** Alarm Overtime Set / **** 2.2 - Alarms - Alarm Generation **** Alarm Overtime Set Timer
   // Alarm Overtime Set
   IF "TRUE" THEN
       #OvtSetAlmTimer(I_StartTimer := (#RunSet OR #C_ManualClampCmdSet) AND NOT #I_DetSet AND NOT #I_RunRes,   // "LTimer"
                       I_HoldTimer := (#IO_Modes.LModeSelector.ManualSel AND #CalibratedSet) OR (#OvtSetAlm AND #CalibratedSet) OR NOT #I_SetIntlkOK OR NOT #I_SafetyOk,
                       I_MaxTimerValue := #OvtAlarmSet,
                       O_TimerResult => #OvtSetAlmResult,
                       O_TimerValue => "NotUsedDInt");
   END_IF;
END_REGION

REGION Network 11: **** 2.2 - Alarms - Alarm Generation **** Alarm Overtime Set Timer -- Calculation Warning/Alarm Time
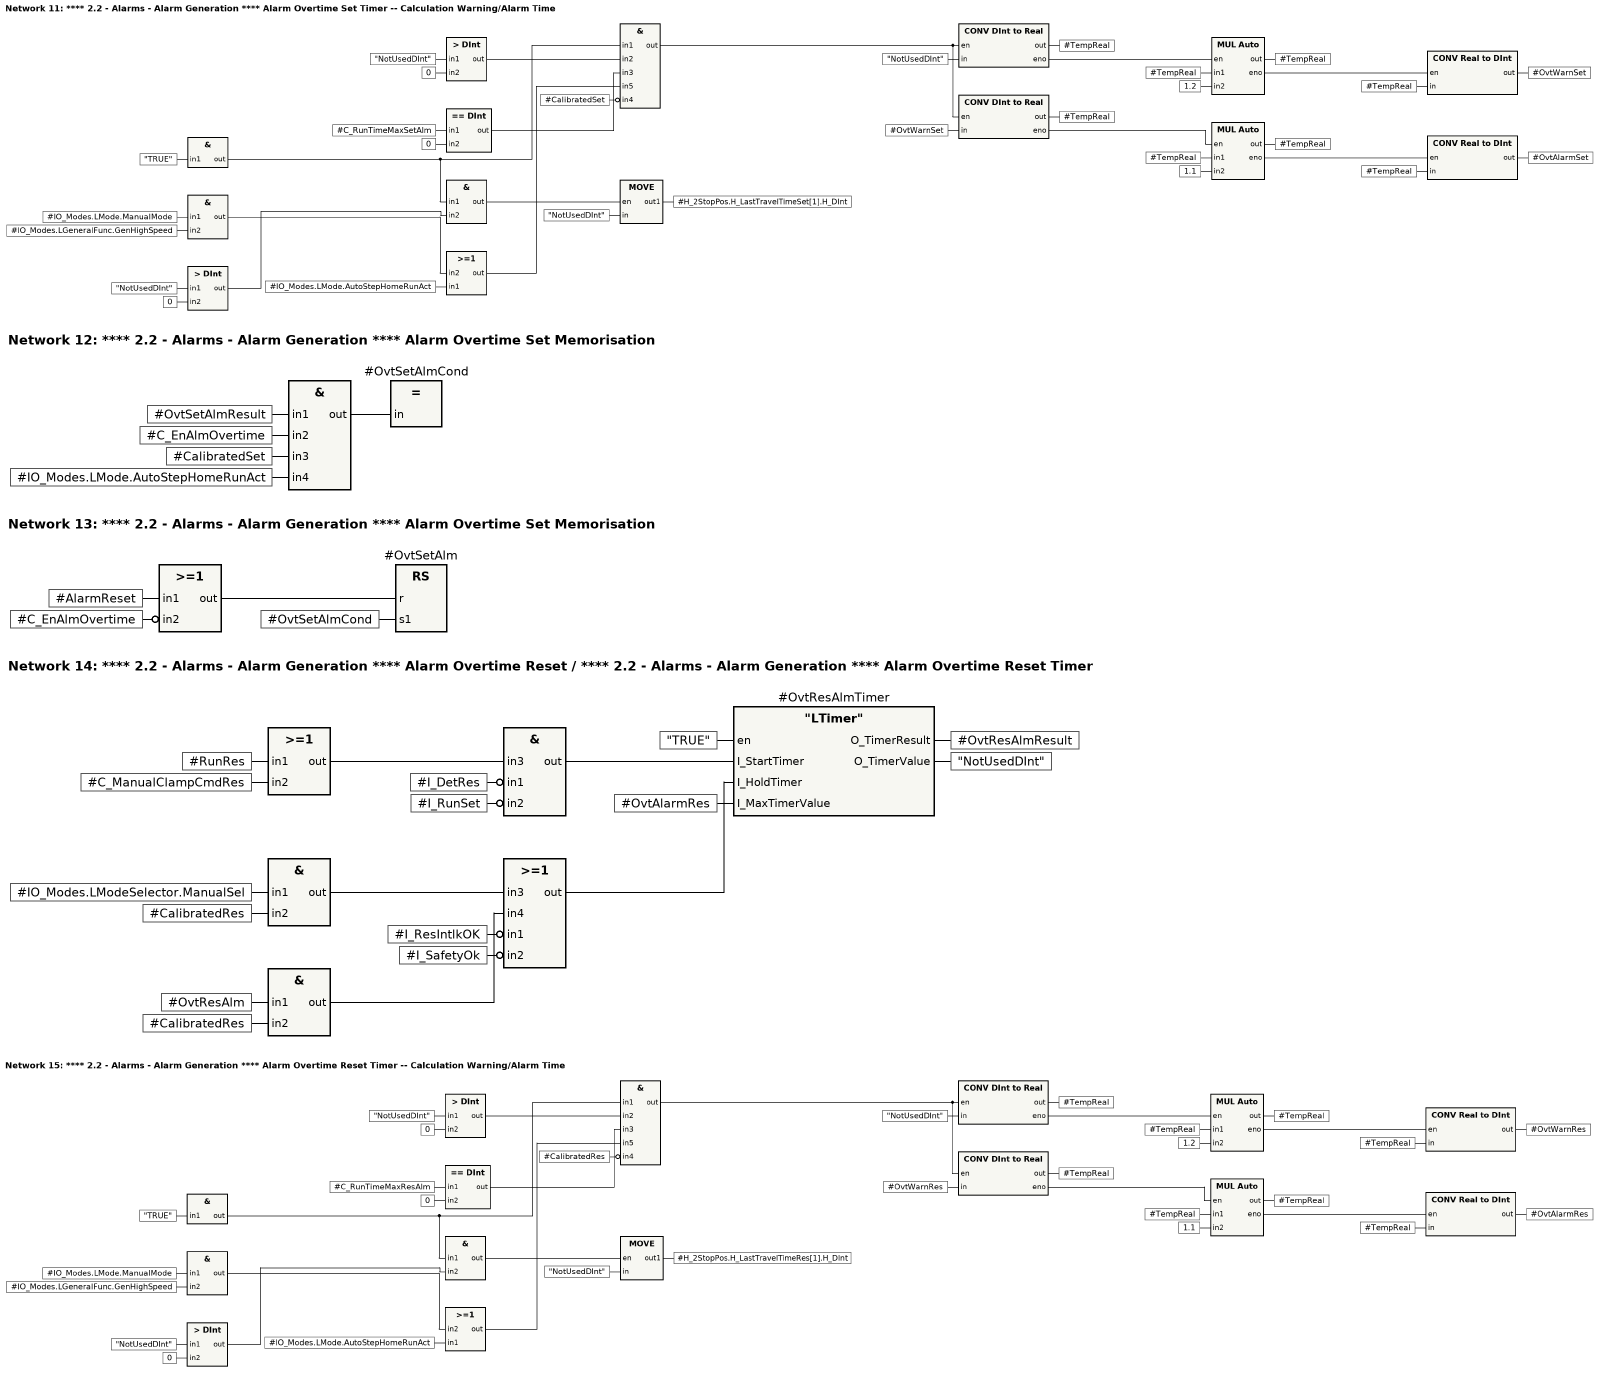
   IF "TRUE" AND ("NotUsedDInt" > 0) AND (#C_RunTimeMaxSetAlm = 0) AND ((#IO_Modes.LMode.ManualMode AND #IO_Modes.LGeneralFunc.GenHighSpeed) OR #IO_Modes.LMode.AutoStepHomeRunAct) AND NOT #CalibratedSet THEN
       #TempReal := DINT_TO_REAL("NotUsedDInt");
       #TempReal := #TempReal * 1.2;
       #OvtWarnSet := REAL_TO_DINT(#TempReal);
       #TempReal := DINT_TO_REAL(#OvtWarnSet);
       #TempReal := #TempReal * 1.1;
       #OvtAlarmSet := REAL_TO_DINT(#TempReal);
   END_IF;
   IF "TRUE" AND ("NotUsedDInt" > 0) THEN #H_2StopPos.H_LastTravelTimeSet[1].H_DInt := "NotUsedDInt"; END_IF;
END_REGION

REGION Network 12: **** 2.2 - Alarms - Alarm Generation **** Alarm Overtime Set Memorisation
   // Alarm Overtime Set Memorisation
   #OvtSetAlmCond := #OvtSetAlmResult AND #C_EnAlmOvertime AND #CalibratedSet AND #IO_Modes.LMode.AutoStepHomeRunAct;
END_REGION

REGION Network 13: **** 2.2 - Alarms - Alarm Generation **** Alarm Overtime Set Memorisation
   // Alarm Overtime Set Memorisation
   IF #AlarmReset OR NOT #C_EnAlmOvertime THEN
       #OvtSetAlm := FALSE;   // RS flip-flop
   END_IF;
   IF #OvtSetAlmCond THEN #OvtSetAlm := TRUE; END_IF;
END_REGION

REGION Network 14: **** 2.2 - Alarms - Alarm Generation **** Alarm Overtime Reset / **** 2.2 - Alarms - Alarm Generation **** Alarm Overtime Reset Timer
   // Alarm Overtime Reset
   IF "TRUE" THEN
       #OvtResAlmTimer(I_StartTimer := (#RunRes OR #C_ManualClampCmdRes) AND NOT #I_DetRes AND NOT #I_RunSet,   // "LTimer"
                       I_HoldTimer := (#IO_Modes.LModeSelector.ManualSel AND #CalibratedRes) OR (#OvtResAlm AND #CalibratedRes) OR NOT #I_ResIntlkOK OR NOT #I_SafetyOk,
                       I_MaxTimerValue := #OvtAlarmRes,
                       O_TimerResult => #OvtResAlmResult,
                       O_TimerValue => "NotUsedDInt");
   END_IF;
END_REGION

REGION Network 15: **** 2.2 - Alarms - Alarm Generation **** Alarm Overtime Reset Timer -- Calculation Warning/Alarm Time
   IF "TRUE" AND ("NotUsedDInt" > 0) AND (#C_RunTimeMaxResAlm = 0) AND ((#IO_Modes.LMode.ManualMode AND #IO_Modes.LGeneralFunc.GenHighSpeed) OR #IO_Modes.LMode.AutoStepHomeRunAct) AND NOT #CalibratedRes THEN
       #TempReal := DINT_TO_REAL("NotUsedDInt");
       #TempReal := #TempReal * 1.2;
       #OvtWarnRes := REAL_TO_DINT(#TempReal);
       #TempReal := DINT_TO_REAL(#OvtWarnRes);
       #TempReal := #TempReal * 1.1;
       #OvtAlarmRes := REAL_TO_DINT(#TempReal);
   END_IF;
   IF "TRUE" AND ("NotUsedDInt" > 0) THEN #H_2StopPos.H_LastTravelTimeRes[1].H_DInt := "NotUsedDInt"; END_IF;
END_REGION

REGION Network 16: **** 2.2 - Alarms - Alarm Generation **** Alarm Overtime Reset Memorisation
   // Alarm Overtime Reset  Memorisation
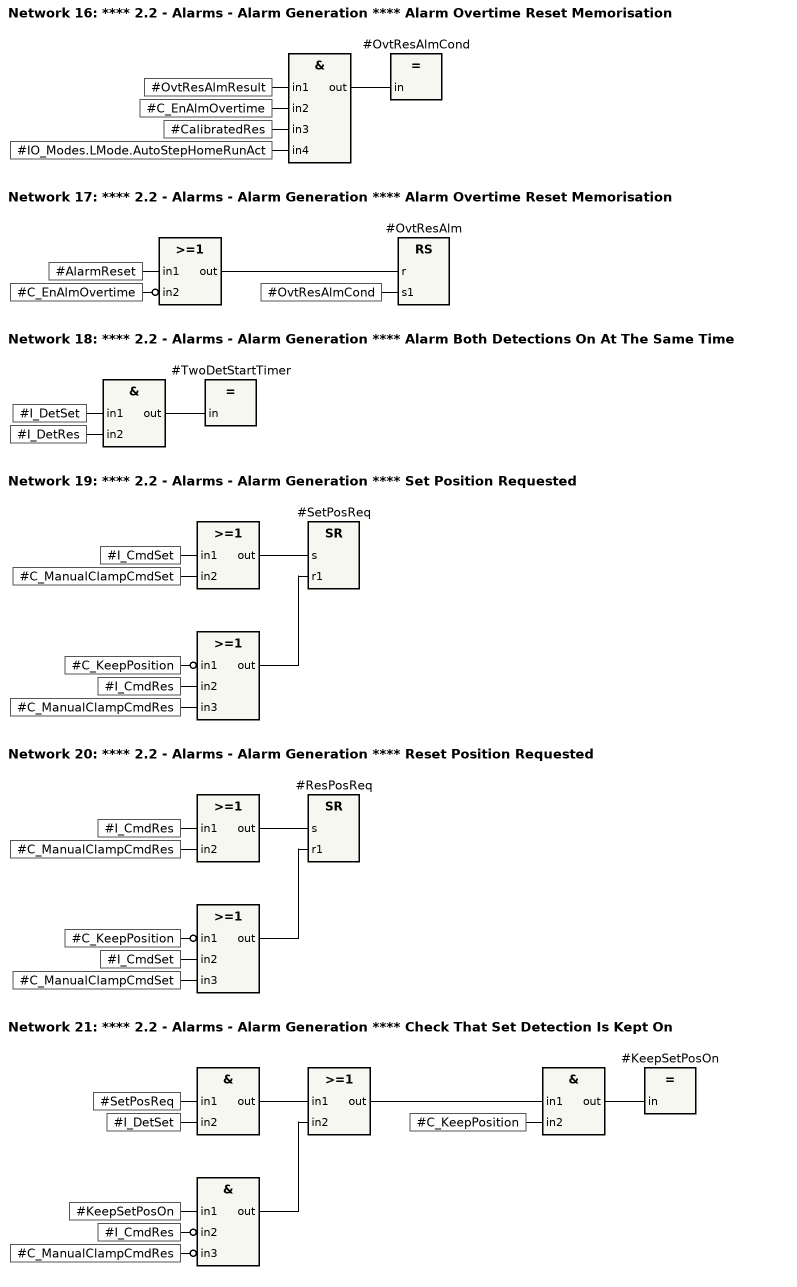
   #OvtResAlmCond := #OvtResAlmResult AND #C_EnAlmOvertime AND #CalibratedRes AND #IO_Modes.LMode.AutoStepHomeRunAct;
END_REGION

REGION Network 17: **** 2.2 - Alarms - Alarm Generation **** Alarm Overtime Reset Memorisation
   // Alarm Overtime Reset  Memorisation
   IF #AlarmReset OR NOT #C_EnAlmOvertime THEN
       #OvtResAlm := FALSE;   // RS flip-flop
   END_IF;
   IF #OvtResAlmCond THEN #OvtResAlm := TRUE; END_IF;
END_REGION

REGION Network 18: **** 2.2 - Alarms - Alarm Generation **** Alarm Both Detections On At The Same Time
   // Alarm Both Detections On At The Same Time
   #TwoDetStartTimer := #I_DetSet AND #I_DetRes;
END_REGION

REGION Network 19: **** 2.2 - Alarms - Alarm Generation **** Set Position Requested
   // Set Position Requested
   IF #I_CmdSet OR #C_ManualClampCmdSet THEN
       #SetPosReq := TRUE;   // SR flip-flop
   END_IF;
   IF NOT #C_KeepPosition OR #I_CmdRes OR #C_ManualClampCmdRes THEN #SetPosReq := FALSE; END_IF;
END_REGION

REGION Network 20: **** 2.2 - Alarms - Alarm Generation **** Reset Position Requested
   // Reset  Position Requested
   IF #I_CmdRes OR #C_ManualClampCmdRes THEN
       #ResPosReq := TRUE;   // SR flip-flop
   END_IF;
   IF NOT #C_KeepPosition OR #I_CmdSet OR #C_ManualClampCmdSet THEN #ResPosReq := FALSE; END_IF;
END_REGION

REGION Network 21: **** 2.2 - Alarms - Alarm Generation **** Check That Set Detection Is Kept On
   // Check That Set Detection Is Kept On
   #KeepSetPosOn := ((#SetPosReq AND #I_DetSet) OR (#KeepSetPosOn AND NOT #I_CmdRes AND NOT #C_ManualClampCmdRes)) AND #C_KeepPosition;
END_REGION

REGION Network 22: **** 2.2 - Alarms - Alarm Generation **** Check That Reset Detection Is Kept On
   // Check That Reset  Detection Is Kept On
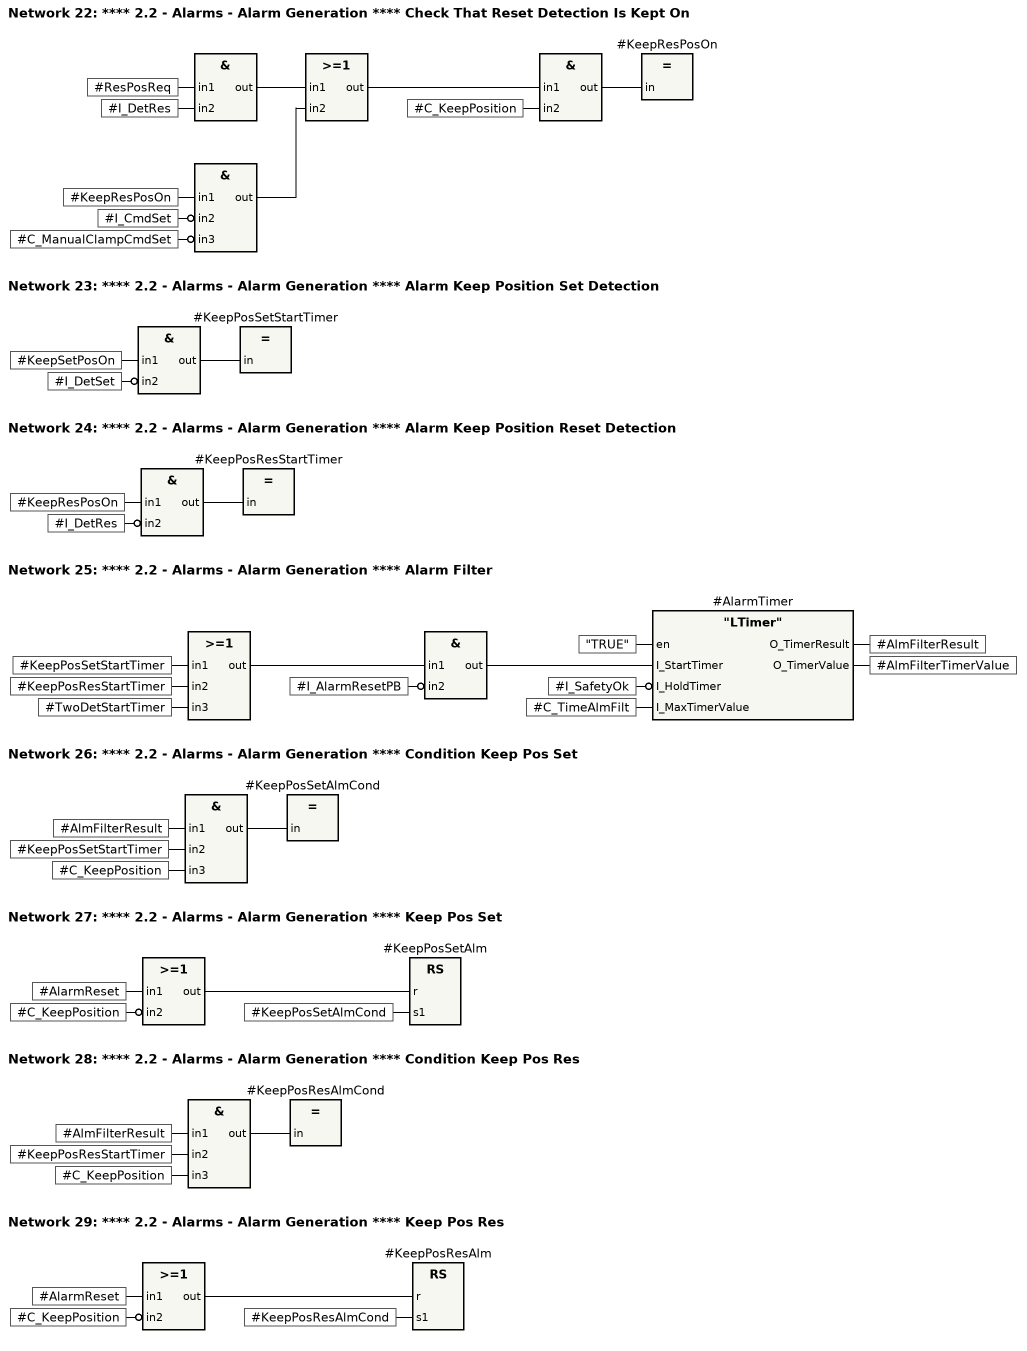
   #KeepResPosOn := ((#ResPosReq AND #I_DetRes) OR (#KeepResPosOn AND NOT #I_CmdSet AND NOT #C_ManualClampCmdSet)) AND #C_KeepPosition;
END_REGION

REGION Network 23: **** 2.2 - Alarms - Alarm Generation **** Alarm Keep Position Set Detection
   // Alarm keep Position Set Detection
   #KeepPosSetStartTimer := #KeepSetPosOn AND NOT #I_DetSet;
END_REGION

REGION Network 24: **** 2.2 - Alarms - Alarm Generation **** Alarm Keep Position Reset Detection
   // Alarm Keep Position Reset  Detection
   #KeepPosResStartTimer := #KeepResPosOn AND NOT #I_DetRes;
END_REGION

REGION Network 25: **** 2.2 - Alarms - Alarm Generation **** Alarm Filter
   // Alarm Filter
   IF "TRUE" THEN
       #AlarmTimer(I_StartTimer := (#KeepPosSetStartTimer OR #KeepPosResStartTimer OR #TwoDetStartTimer) AND NOT #I_AlarmResetPB,   // "LTimer"
                   I_HoldTimer := NOT #I_SafetyOk,
                   I_MaxTimerValue := #C_TimeAlmFilt,
                   O_TimerResult => #AlmFilterResult,
                   O_TimerValue => #AlmFilterTimerValue);
   END_IF;
END_REGION

REGION Network 26: **** 2.2 - Alarms - Alarm Generation **** Condition Keep Pos Set
   // Condition Keep Pos Set
   #KeepPosSetAlmCond := #AlmFilterResult AND #KeepPosSetStartTimer AND #C_KeepPosition;
END_REGION

REGION Network 27: **** 2.2 - Alarms - Alarm Generation **** Keep Pos Set
   // Keep Pos Set
   IF #AlarmReset OR NOT #C_KeepPosition THEN
       #KeepPosSetAlm := FALSE;   // RS flip-flop
   END_IF;
   IF #KeepPosSetAlmCond THEN #KeepPosSetAlm := TRUE; END_IF;
END_REGION

REGION Network 28: **** 2.2 - Alarms - Alarm Generation **** Condition Keep Pos Res
   // Condition Keep Pos Res
   #KeepPosResAlmCond := #AlmFilterResult AND #KeepPosResStartTimer AND #C_KeepPosition;
END_REGION

REGION Network 29: **** 2.2 - Alarms - Alarm Generation **** Keep Pos Res
   // Keep Pos Res
   IF #AlarmReset OR NOT #C_KeepPosition THEN
       #KeepPosResAlm := FALSE;   // RS flip-flop
   END_IF;
   IF #KeepPosResAlmCond THEN #KeepPosResAlm := TRUE; END_IF;
END_REGION

REGION Network 30: **** 2.2 - Alarms - Alarm Generation **** 2 Detection Alarm
   // 2 Detection Alarm
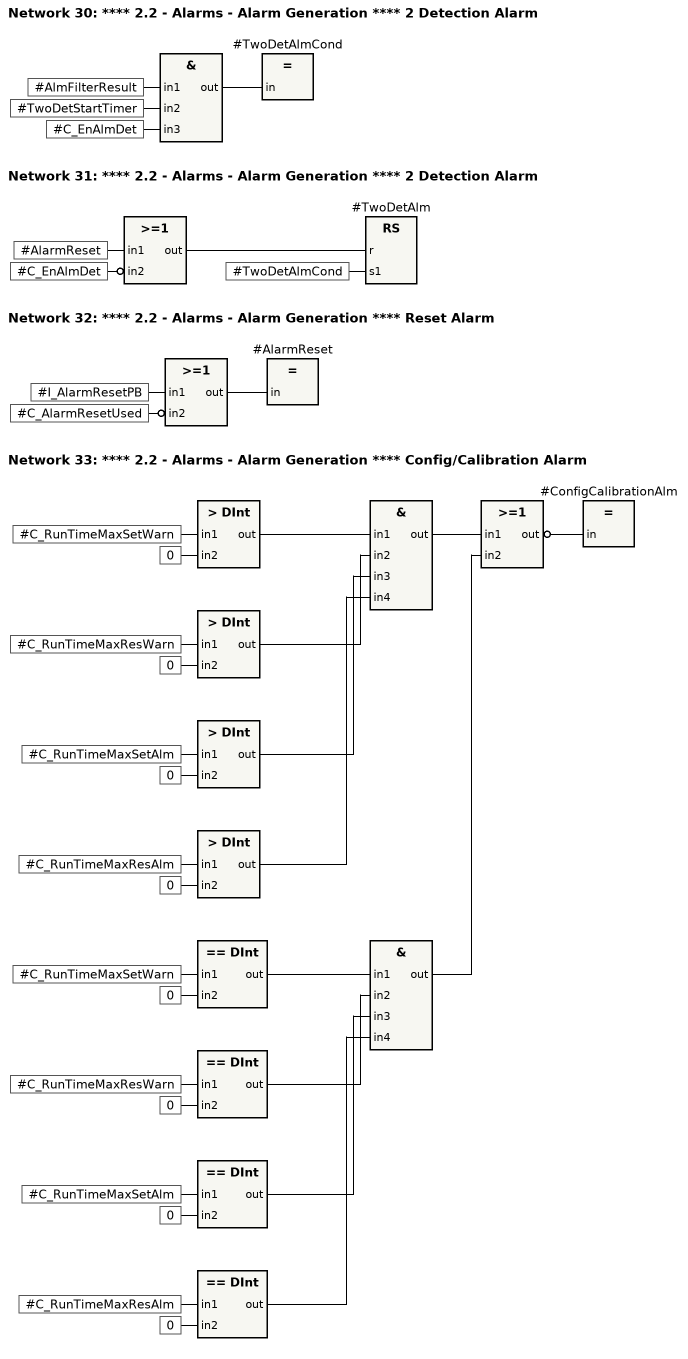
   #TwoDetAlmCond := #AlmFilterResult AND #TwoDetStartTimer AND #C_EnAlmDet;
END_REGION

REGION Network 31: **** 2.2 - Alarms - Alarm Generation **** 2 Detection Alarm
   // 2 Detection Alarm
   IF #AlarmReset OR NOT #C_EnAlmDet THEN
       #TwoDetAlm := FALSE;   // RS flip-flop
   END_IF;
   IF #TwoDetAlmCond THEN #TwoDetAlm := TRUE; END_IF;
END_REGION

REGION Network 32: **** 2.2 - Alarms - Alarm Generation **** Reset Alarm
   // Reset  Alarm
   #AlarmReset := #I_AlarmResetPB OR NOT #C_AlarmResetUsed;
END_REGION

REGION Network 33: **** 2.2 - Alarms - Alarm Generation **** Config/Calibration Alarm
   #ConfigCalibrationAlm := NOT (((#C_RunTimeMaxSetWarn > 0) AND (#C_RunTimeMaxResWarn > 0) AND (#C_RunTimeMaxSetAlm > 0) AND (#C_RunTimeMaxResAlm > 0)) OR ((#C_RunTimeMaxSetWarn = 0) AND (#C_RunTimeMaxResWarn = 0) AND (#C_RunTimeMaxSetAlm = 0) AND (#C_RunTimeMaxResAlm = 0)));
END_REGION

REGION Network 34: **** 2.2 - Alarms - Alarm Generation **** Calibration Warning
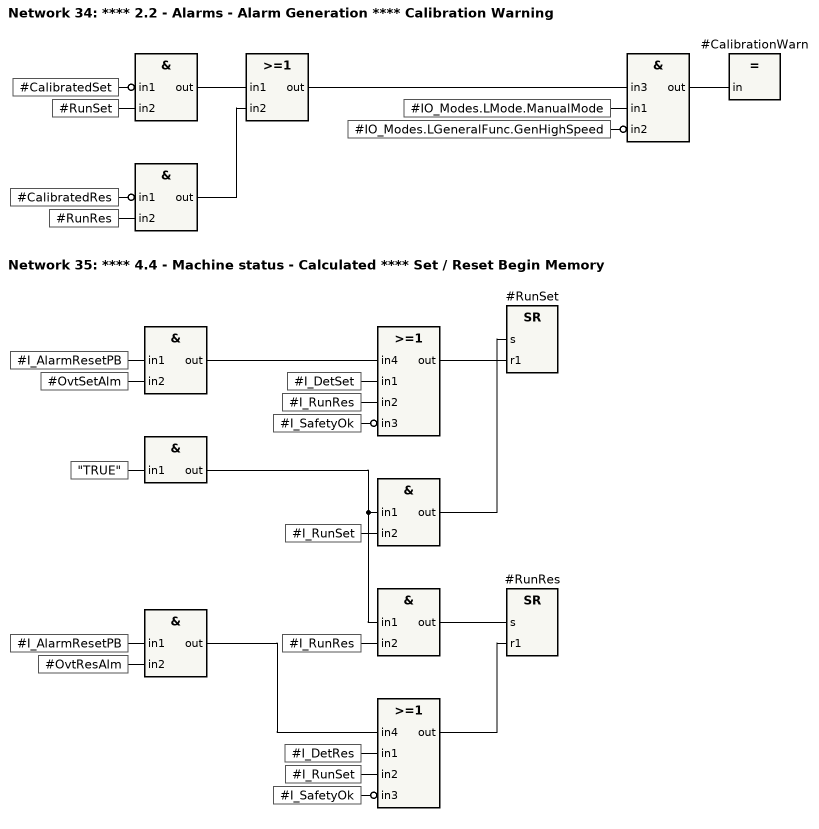
   #CalibrationWarn := ((NOT #CalibratedSet AND #RunSet) OR (NOT #CalibratedRes AND #RunRes)) AND #IO_Modes.LMode.ManualMode AND NOT #IO_Modes.LGeneralFunc.GenHighSpeed;
END_REGION

REGION Network 35: **** 4.4 - Machine status - Calculated **** Set / Reset Begin Memory
   // Set / Reset Begin Memory / Delay of Set Position
   IF "TRUE" AND #I_RunSet THEN
       #RunSet := TRUE;   // SR flip-flop
   END_IF;
   IF (#I_AlarmResetPB AND #OvtSetAlm) OR #I_DetSet OR #I_RunRes OR NOT #I_SafetyOk THEN
       #RunSet := FALSE;
   END_IF;
   IF "TRUE" AND #I_RunRes THEN
       #RunRes := TRUE;   // SR flip-flop
   END_IF;
   IF (#I_AlarmResetPB AND #OvtResAlm) OR #I_DetRes OR #I_RunSet OR NOT #I_SafetyOk THEN
       #RunRes := FALSE;
   END_IF;
END_REGION

REGION Network 36: **** 4.6 - Machine Status - Indication **** Icon Animation / **** 4.6 - Machine status - Indication **** Icon Animation
   // Icon Animation
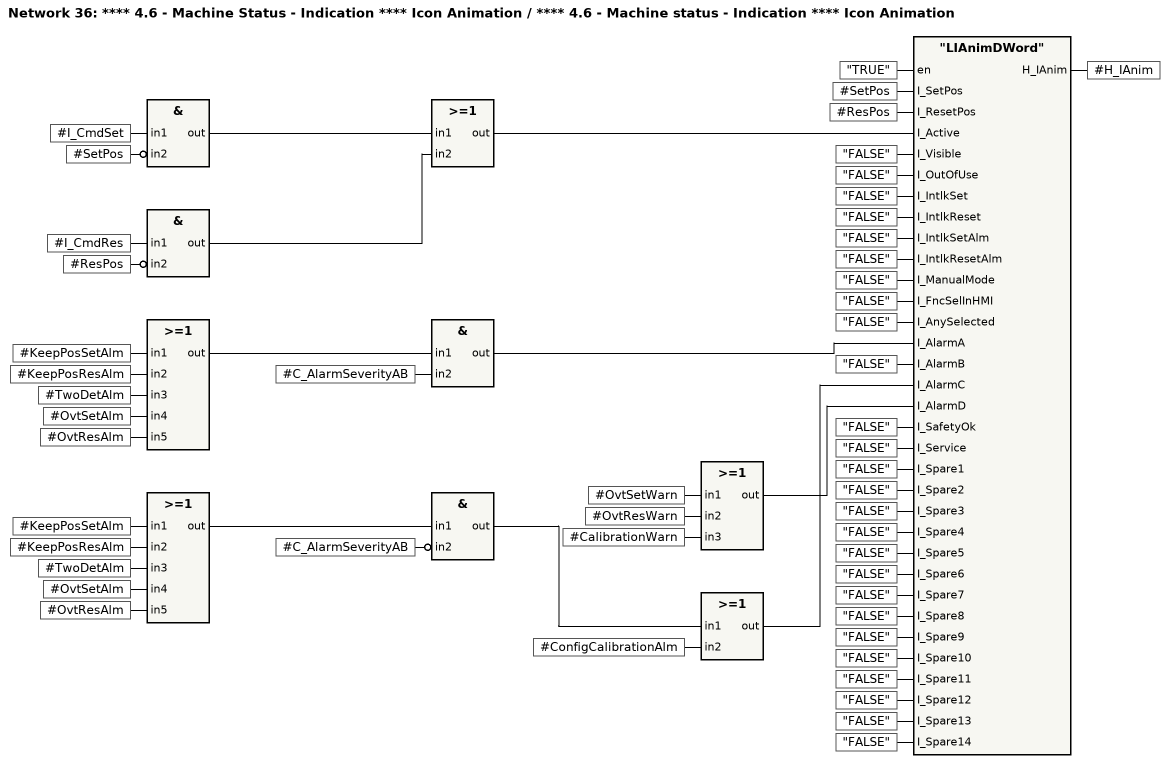
   IF "TRUE" THEN
       "LIAnimDWord"(I_SetPos := #SetPos,
                     I_ResetPos := #ResPos,
                     I_Active := (#I_CmdSet AND NOT #SetPos) OR (#I_CmdRes AND NOT #ResPos),
                     I_Visible := "FALSE",
                     I_OutOfUse := "FALSE",
                     I_IntlkSet := "FALSE",
                     I_IntlkReset := "FALSE",
                     I_IntlkSetAlm := "FALSE",
                     I_IntlkResetAlm := "FALSE",
                     I_ManualMode := "FALSE",
                     I_FncSelInHMI := "FALSE",
                     I_AnySelected := "FALSE",
                     I_AlarmA := (#KeepPosSetAlm OR #KeepPosResAlm OR #TwoDetAlm OR #OvtSetAlm OR #OvtResAlm) AND #C_AlarmSeverityAB,
                     I_AlarmB := "FALSE",
                     I_AlarmC := ((#KeepPosSetAlm OR #KeepPosResAlm OR #TwoDetAlm OR #OvtSetAlm OR #OvtResAlm) AND NOT #C_AlarmSeverityAB) OR #ConfigCalibrationAlm,
                     I_AlarmD := #OvtSetWarn OR #OvtResWarn OR #CalibrationWarn,
                     I_SafetyOk := "FALSE",
                     I_Service := "FALSE",
                     I_Spare1 := "FALSE",
                     I_Spare2 := "FALSE",
                     I_Spare3 := "FALSE",
                     I_Spare4 := "FALSE",
                     I_Spare5 := "FALSE",
                     I_Spare6 := "FALSE",
                     I_Spare7 := "FALSE",
                     I_Spare8 := "FALSE",
                     I_Spare9 := "FALSE",
                     I_Spare10 := "FALSE",
                     I_Spare11 := "FALSE",
                     I_Spare12 := "FALSE",
                     I_Spare13 := "FALSE",
                     I_Spare14 := "FALSE",
                     H_IAnim => #H_IAnim);
   END_IF;
END_REGION

REGION Network 37: **** 4.6 - Machine Status - Indication **** Animation / **** 4.6 - Machine status - Indication **** Animation
   // Animation
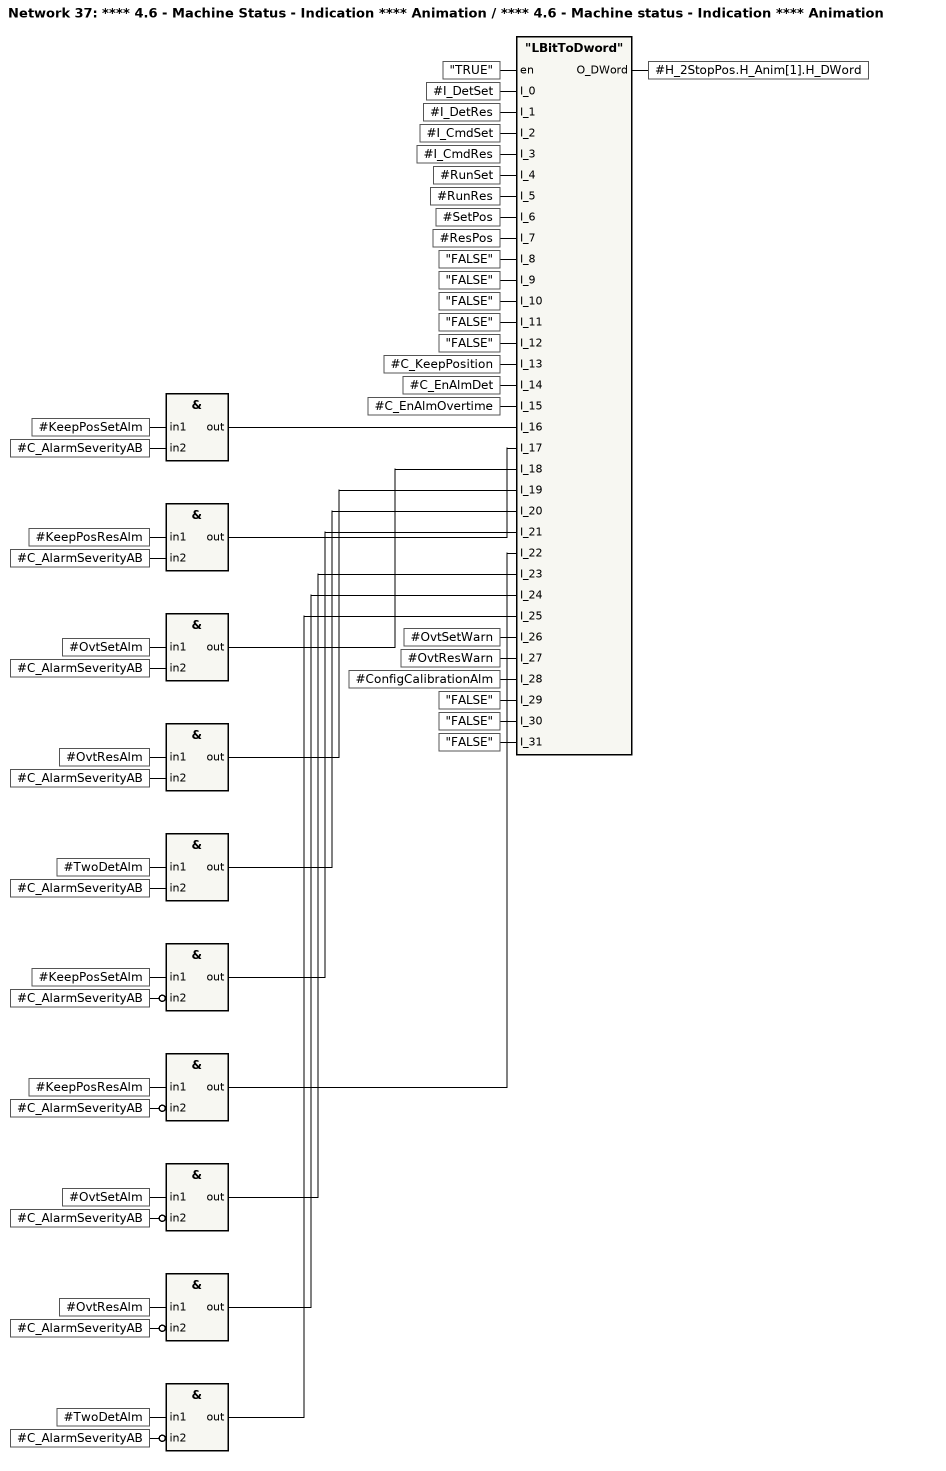
   IF "TRUE" THEN
       "LBitToDword"(I_0 := #I_DetSet,
                     I_1 := #I_DetRes,
                     I_2 := #I_CmdSet,
                     I_3 := #I_CmdRes,
                     I_4 := #RunSet,
                     I_5 := #RunRes,
                     I_6 := #SetPos,
                     I_7 := #ResPos,
                     I_8 := "FALSE",
                     I_9 := "FALSE",
                     I_10 := "FALSE",
                     I_11 := "FALSE",
                     I_12 := "FALSE",
                     I_13 := #C_KeepPosition,
                     I_14 := #C_EnAlmDet,
                     I_15 := #C_EnAlmOvertime,
                     I_16 := #KeepPosSetAlm AND #C_AlarmSeverityAB,
                     I_17 := #KeepPosResAlm AND #C_AlarmSeverityAB,
                     I_18 := #OvtSetAlm AND #C_AlarmSeverityAB,
                     I_19 := #OvtResAlm AND #C_AlarmSeverityAB,
                     I_20 := #TwoDetAlm AND #C_AlarmSeverityAB,
                     I_21 := #KeepPosSetAlm AND NOT #C_AlarmSeverityAB,
                     I_22 := #KeepPosResAlm AND NOT #C_AlarmSeverityAB,
                     I_23 := #OvtSetAlm AND NOT #C_AlarmSeverityAB,
                     I_24 := #OvtResAlm AND NOT #C_AlarmSeverityAB,
                     I_25 := #TwoDetAlm AND NOT #C_AlarmSeverityAB,
                     I_26 := #OvtSetWarn,
                     I_27 := #OvtResWarn,
                     I_28 := #ConfigCalibrationAlm,
                     I_29 := "FALSE",
                     I_30 := "FALSE",
                     I_31 := "FALSE",
                     O_DWord => #H_2StopPos.H_Anim[1].H_DWord);
   END_IF;
END_REGION

REGION Network 38: **** 4.6 - Machine status - Indication **** Animation
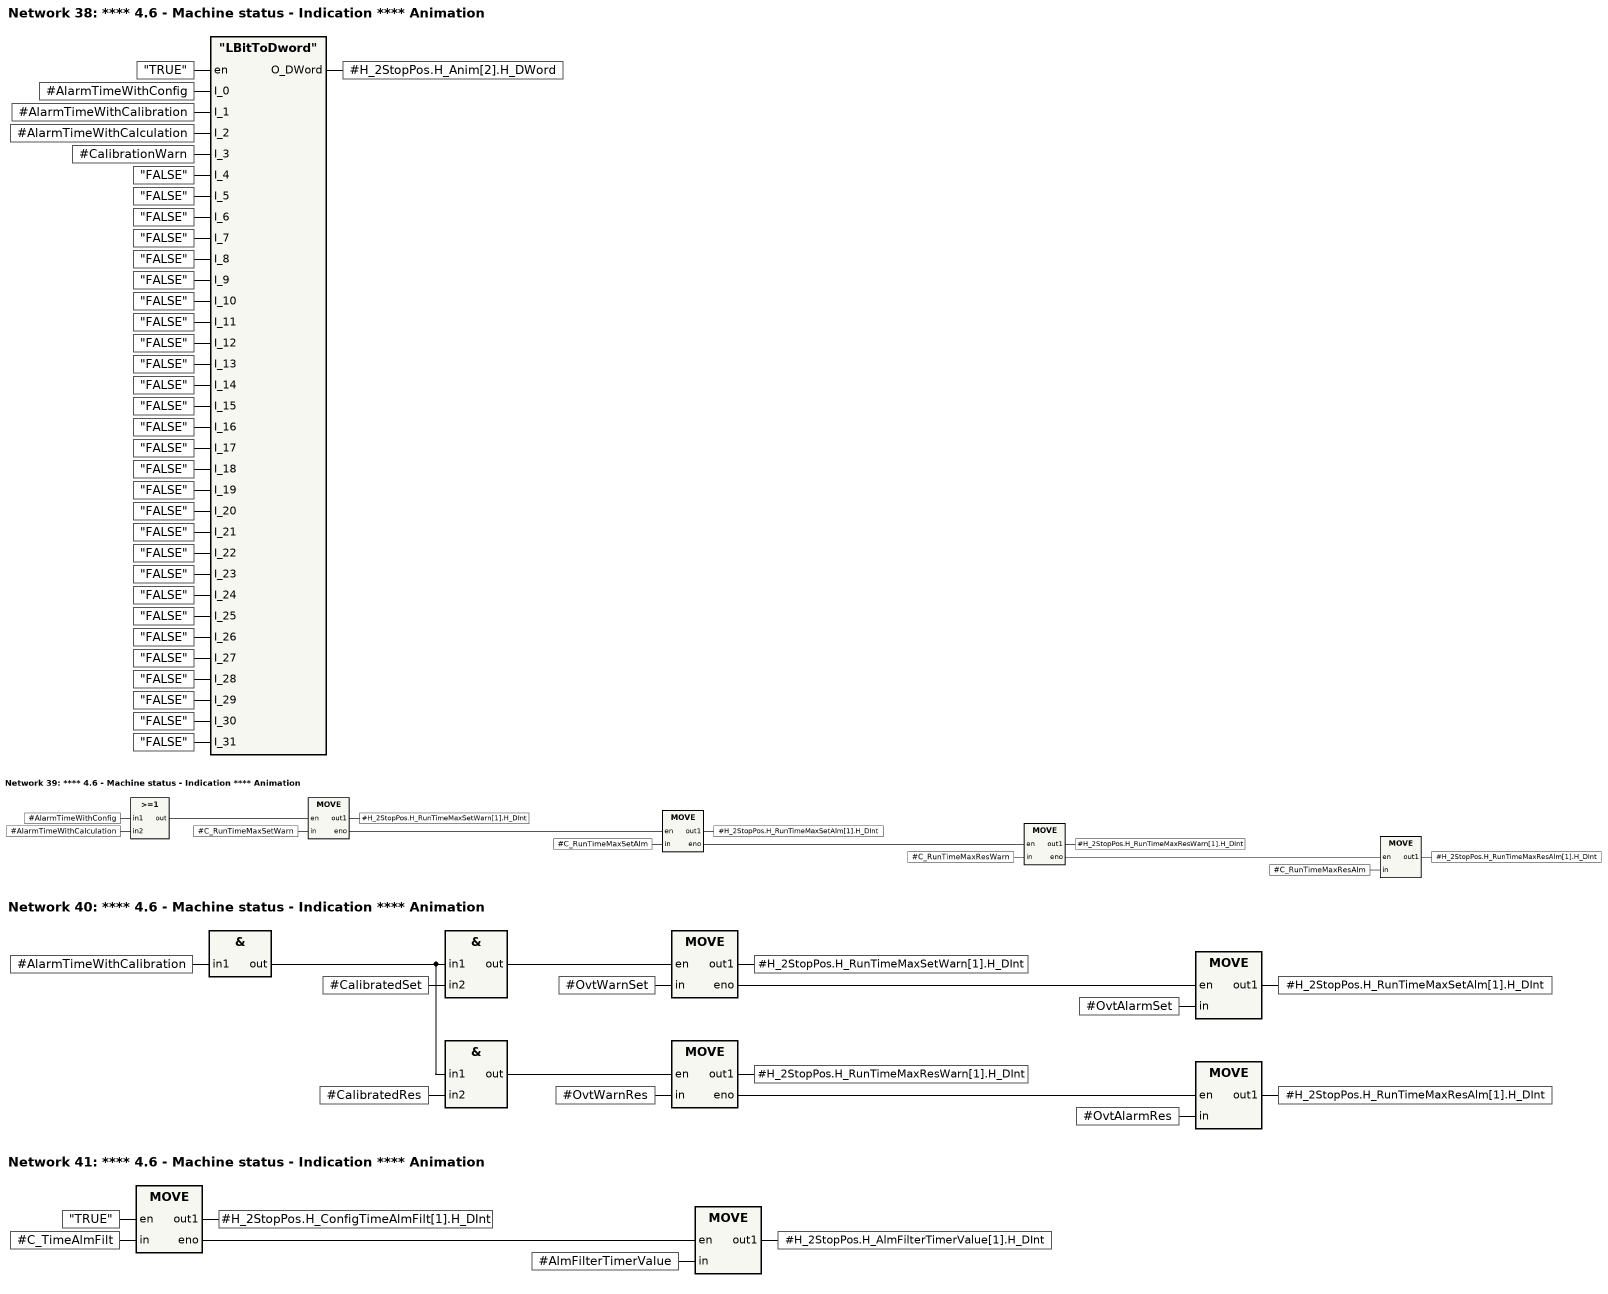
   IF "TRUE" THEN
       "LBitToDword"(I_0 := #AlarmTimeWithConfig,
                     I_1 := #AlarmTimeWithCalibration,
                     I_2 := #AlarmTimeWithCalculation,
                     I_3 := #CalibrationWarn,
                     I_4 := "FALSE",
                     I_5 := "FALSE",
                     I_6 := "FALSE",
                     I_7 := "FALSE",
                     I_8 := "FALSE",
                     I_9 := "FALSE",
                     I_10 := "FALSE",
                     I_11 := "FALSE",
                     I_12 := "FALSE",
                     I_13 := "FALSE",
                     I_14 := "FALSE",
                     I_15 := "FALSE",
                     I_16 := "FALSE",
                     I_17 := "FALSE",
                     I_18 := "FALSE",
                     I_19 := "FALSE",
                     I_20 := "FALSE",
                     I_21 := "FALSE",
                     I_22 := "FALSE",
                     I_23 := "FALSE",
                     I_24 := "FALSE",
                     I_25 := "FALSE",
                     I_26 := "FALSE",
                     I_27 := "FALSE",
                     I_28 := "FALSE",
                     I_29 := "FALSE",
                     I_30 := "FALSE",
                     I_31 := "FALSE",
                     O_DWord => #H_2StopPos.H_Anim[2].H_DWord);
   END_IF;
END_REGION

REGION Network 39: **** 4.6 - Machine status - Indication **** Animation
   IF #AlarmTimeWithConfig OR #AlarmTimeWithCalculation THEN
       #H_2StopPos.H_RunTimeMaxSetWarn[1].H_DInt := #C_RunTimeMaxSetWarn;
       #H_2StopPos.H_RunTimeMaxSetAlm[1].H_DInt := #C_RunTimeMaxSetAlm;
       #H_2StopPos.H_RunTimeMaxResWarn[1].H_DInt := #C_RunTimeMaxResWarn;
       #H_2StopPos.H_RunTimeMaxResAlm[1].H_DInt := #C_RunTimeMaxResAlm;
   END_IF;
END_REGION

REGION Network 40: **** 4.6 - Machine status - Indication **** Animation
   IF #AlarmTimeWithCalibration AND #CalibratedSet THEN
       #H_2StopPos.H_RunTimeMaxSetWarn[1].H_DInt := #OvtWarnSet;
       #H_2StopPos.H_RunTimeMaxSetAlm[1].H_DInt := #OvtAlarmSet;
   END_IF;
   IF #AlarmTimeWithCalibration AND #CalibratedRes THEN
       #H_2StopPos.H_RunTimeMaxResWarn[1].H_DInt := #OvtWarnRes;
       #H_2StopPos.H_RunTimeMaxResAlm[1].H_DInt := #OvtAlarmRes;
   END_IF;
END_REGION

REGION Network 41: **** 4.6 - Machine status - Indication **** Animation
   IF "TRUE" THEN
       #H_2StopPos.H_ConfigTimeAlmFilt[1].H_DInt := #C_TimeAlmFilt;
       #H_2StopPos.H_AlmFilterTimerValue[1].H_DInt := #AlmFilterTimerValue;
   END_IF;
END_REGION

REGION Network 42: **** 5.2 - Equations - Flow Equations **** Set Position
   // Set Position
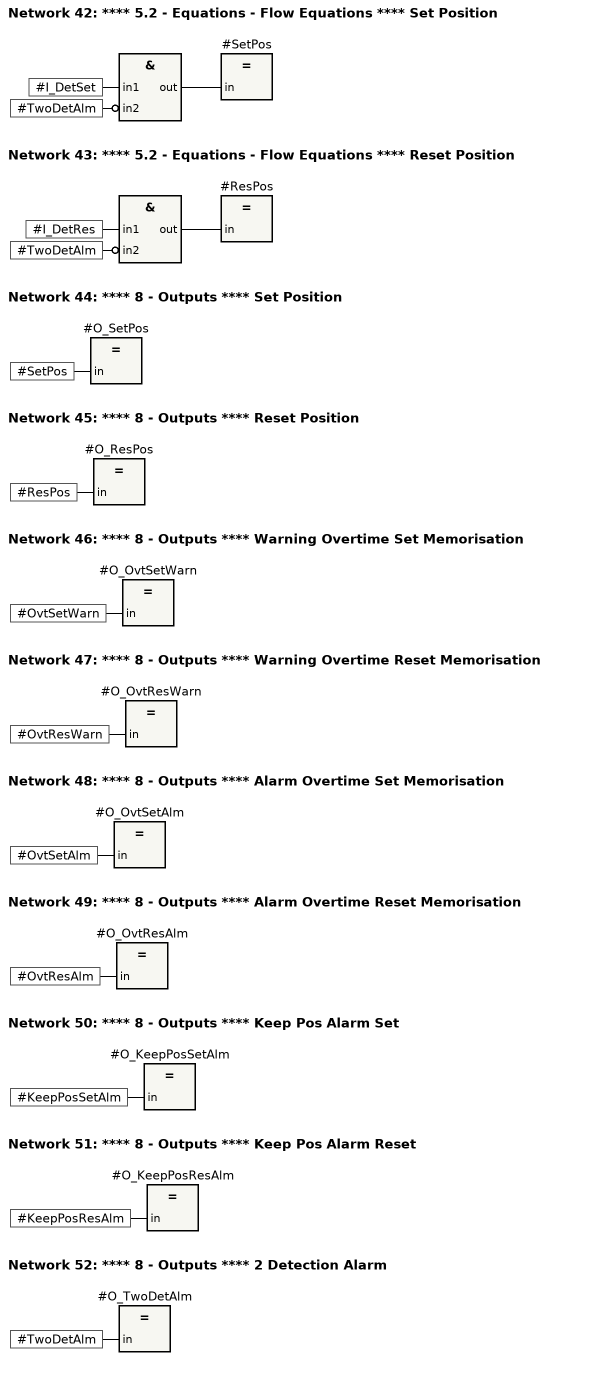
   #SetPos := #I_DetSet AND NOT #TwoDetAlm;
END_REGION

REGION Network 43: **** 5.2 - Equations - Flow Equations **** Reset Position
   // Reset  Position
   #ResPos := #I_DetRes AND NOT #TwoDetAlm;
END_REGION

REGION Network 44: **** 8 - Outputs **** Set Position
   // Set Position
   #O_SetPos := #SetPos;
END_REGION

REGION Network 45: **** 8 - Outputs **** Reset Position
   // Reset  Position
   #O_ResPos := #ResPos;
END_REGION

REGION Network 46: **** 8 - Outputs **** Warning Overtime Set Memorisation
   // Warning Overtime Set Memorisation
   #O_OvtSetWarn := #OvtSetWarn;
END_REGION

REGION Network 47: **** 8 - Outputs **** Warning Overtime Reset Memorisation
   // Warning Overtime Reset  Memorisation
   #O_OvtResWarn := #OvtResWarn;
END_REGION

REGION Network 48: **** 8 - Outputs **** Alarm Overtime Set Memorisation
   // Alarm Overtime Set Memorisation
   #O_OvtSetAlm := #OvtSetAlm;
END_REGION

REGION Network 49: **** 8 - Outputs **** Alarm Overtime Reset Memorisation
   // Alarm Overtime Reset  Memorisation
   #O_OvtResAlm := #OvtResAlm;
END_REGION

REGION Network 50: **** 8 - Outputs **** Keep Pos Alarm Set
   // Keep Pos Alarm Set
   #O_KeepPosSetAlm := #KeepPosSetAlm;
END_REGION

REGION Network 51: **** 8 - Outputs **** Keep Pos Alarm Reset
   // Keep Pos Alarm Reset
   #O_KeepPosResAlm := #KeepPosResAlm;
END_REGION

REGION Network 52: **** 8 - Outputs **** 2 Detection Alarm
   // 2 Detection Alarm
   #O_TwoDetAlm := #TwoDetAlm;
END_REGION

REGION Network 53: **** 8 - Outputs **** Config/Calibration Alarm
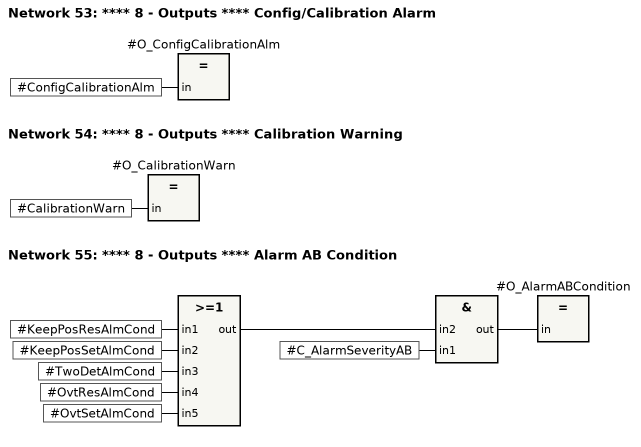
   #O_ConfigCalibrationAlm := #ConfigCalibrationAlm;
END_REGION

REGION Network 54: **** 8 - Outputs **** Calibration Warning
   #O_CalibrationWarn := #CalibrationWarn;
END_REGION

REGION Network 55: **** 8 - Outputs **** Alarm AB Condition
   // Alarm AB Condition
   #O_AlarmABCondition := (#KeepPosResAlmCond OR #KeepPosSetAlmCond OR #TwoDetAlmCond OR #OvtResAlmCond OR #OvtSetAlmCond) AND #C_AlarmSeverityAB;
END_REGION
END_FUNCTION_BLOCK

